LIN {X 0.037,Y -167.701,Z 831.356,A 0.000,B 0.000,C 90.000,E1 244.101} C_DIS
LIN {X 0.050,Y -166.387,Z 831.347,A 0.000,B 0.000,C 90.000,E1 242.359} C_DIS
LIN {X 0.041,Y -163.114,Z 831.327,A 0.000,B 0.000,C 90.000,E1 238.869} C_DIS
LIN {X 0.091,Y -161.064,Z 831.313,A 0.000,B 0.000,C 90.000,E1 236.215} C_DIS
LIN {X -0.021,Y -157.797,Z 831.293,A 0.000,B 0.000,C 90.000,E1 232.718} C_DIS
LIN {X 0.017,Y -155.833,Z 831.278,A 0.000,B 0.000,C 90.000,E1 230.033} C_DIS
LIN {X -0.026,Y -152.084,Z 831.253,A 0.000,B 0.000,C 90.000,E1 225.567} C_DIS
LIN {X -0.007,Y -150.334,Z 831.238,A 0.000,B 0.000,C 90.000,E1 222.852} C_DIS
LIN {X 0.014,Y -147.073,Z 831.213,A 0.000,B 0.000,C 90.000,E1 218.302} C_DIS
LIN {X -0.083,Y -145.648,Z 831.198,A 0.000,B 0.000,C 90.000,E1 215.598} C_DIS
LIN {X -0.078,Y -143.030,Z 831.172,A 0.000,B 0.000,C 90.000,E1 211.003} C_DIS
LIN {X 0.049,Y -141.656,Z 831.152,A 0.000,B 0.000,C 90.000,E1 207.257} C_DIS
LIN {X -0.032,Y -139.446,Z 831.115,A 0.000,B 0.000,C 90.000,E1 200.791} C_DIS
LIN {X 0.021,Y -139.179,Z 831.105,A 0.000,B 0.000,C 90.000,E1 198.906} C_DIS
LIN {X 0.049,Y -138.320,Z 831.053,A 0.000,B 0.000,C 90.000,E1 189.557} C_DIS
LIN {X 0.058,Y -139.466,Z 831.006,A 0.000,B 0.000,C 90.000,E1 181.146} C_DIS
LIN {X 0.000,Y -141.031,Z 830.975,A 0.000,B 0.000,C 90.000,E1 175.584} C_DIS
LIN {X -0.047,Y -142.398,Z 830.960,A 0.000,B 0.000,C 90.000,E1 172.818} C_DIS
LIN {X 0.016,Y -144.630,Z 830.934,A 0.000,B 0.000,C 90.000,E1 168.173} C_DIS
LIN {X 0.076,Y -147.825,Z 830.909,A 0.000,B 0.000,C 90.000,E1 163.559} C_DIS
LIN {X 0.021,Y -150.518,Z 830.889,A 0.000,B 0.000,C 90.000,E1 159.934} C_DIS
LIN {X 0.041,Y -153.979,Z 830.868,A 0.000,B 0.000,C 90.000,E1 156.305} C_DIS
LIN {X -0.038,Y -157.392,Z 830.849,A 0.000,B 0.000,C 90.000,E1 152.743} C_DIS
LIN {X 0.042,Y -161.596,Z 830.829,A 0.000,B 0.000,C 90.000,E1 149.154} C_DIS
LIN {X -0.086,Y -165.793,Z 830.809,A 0.000,B 0.000,C 90.000,E1 145.674} C_DIS
LIN {X 0.034,Y -170.757,Z 830.790,A 0.000,B 0.000,C 90.000,E1 142.145} C_DIS
LIN {X 0.057,Y -175.628,Z 830.771,A 0.000,B 0.000,C 90.000,E1 138.690} C_DIS
LIN {X -0.074,Y -181.244,Z 830.752,A 0.000,B 0.000,C 90.000,E1 135.324} C_DIS
LIN {X 0.057,Y -186.714,Z 830.733,A 0.000,B 0.000,C 90.000,E1 131.919} C_DIS
LIN {X 0.008,Y -191.313,Z 830.719,A 0.000,B 0.000,C 90.000,E1 129.439} C_DIS
LIN {X -0.064,Y -192.836,Z 830.714,A 0.000,B 0.000,C 90.000,E1 128.543} C_DIS
LIN {X -0.132,Y -292.864,Z 830.714,A 0.000,B 0.000,C 90.000,E1 128.543} C_DIS
LIN {X 0.072,Y -295.448,Z 830.714,A 0.000,B 0.000,C 90.000,E1 128.463} C_DIS
LIN {X -0.036,Y -301.314,Z 830.712,A 0.000,B 0.000,C 90.000,E1 128.141} C_DIS
LIN {X -0.096,Y -304.356,Z 830.710,A 0.000,B 0.000,C 90.000,E1 127.810} C_DIS
LIN {X -0.033,Y -306.345,Z 830.708,A 0.000,B 0.000,C 90.000,E1 127.488} C_DIS
LIN {X 0.087,Y -307.898,Z 830.707,A 0.000,B 0.000,C 90.000,E1 127.156} C_DIS
LIN {X -0.132,Y -309.196,Z 830.705,A 0.000,B 0.000,C 90.000,E1 126.870} C_DIS
LIN {X 0.029,Y -321.363,Z 830.683,A 0.000,B 0.000,C 90.000,E1 122.959} C_DIS
LIN {X -0.104,Y -331.880,Z 830.667,A 0.000,B 0.000,C 90.000,E1 120.129} C_DIS
LIN {X 0.017,Y -343.755,Z 830.652,A 0.000,B 0.000,C 90.000,E1 117.308} C_DIS
LIN {X -0.150,Y -357.097,Z 830.636,A 0.000,B 0.000,C 90.000,E1 114.591} C_DIS
LIN {X -0.166,Y -370.281,Z 830.623,A 0.000,B 0.000,C 90.000,E1 112.206} C_DIS
LIN {X 0.217,Y -384.810,Z 830.610,A 0.000,B 0.000,C 90.000,E1 109.812} C_DIS
LIN {X -0.143,Y -400.790,Z 830.598,A 0.000,B 0.000,C 90.000,E1 107.583} C_DIS
LIN {X -0.242,Y -418.334,Z 830.585,A 0.000,B 0.000,C 90.000,E1 105.371} C_DIS
LIN {X -0.002,Y -437.542,Z 830.573,A 0.000,B 0.000,C 90.000,E1 103.175} C_DIS
LIN {X 0.205,Y -457.699,Z 830.562,A 0.000,B 0.000,C 90.000,E1 101.130} C_DIS
LIN {X 0.102,Y -467.922,Z 830.557,A 0.000,B 0.000,C 90.000,E1 100.197} C_DIS
LIN {X 0.100,Y -469.931,Z 830.555,A 0.000,B 0.000,C 90.000,E1 99.962} C_DIS
LIN {X 0.096,Y -471.458,Z 830.554,A 0.000,B 0.000,C 90.000,E1 99.726} C_DIS
LIN {X -0.129,Y -472.703,Z 830.553,A 0.000,B 0.000,C 90.000,E1 99.500} C_DIS
LIN {X 0.193,Y -473.614,Z 830.551,A 0.000,B 0.000,C 90.000,E1 99.208} C_DIS
LIN {X -0.161,Y -474.606,Z 830.548,A 0.000,B 0.000,C 90.000,E1 98.746} C_DIS
LIN {X 0.031,Y -474.616,Z 830.546,A 0.000,B 0.000,C 90.000,E1 98.219} C_DIS
LIN {X 0.158,Y -473.647,Z 830.543,A 0.000,B 0.000,C 90.000,E1 97.701} C_DIS
LIN {X -0.182,Y -471.537,Z 830.540,A 0.000,B 0.000,C 90.000,E1 97.239} C_DIS
LIN {X -0.007,Y -453.828,Z 830.525,A 0.000,B 0.000,C 90.000,E1 94.416} C_DIS
LIN {X 0.139,Y -443.235,Z 830.514,A 0.000,B 0.000,C 90.000,E1 92.579} C_DIS
LIN {X -0.113,Y -433.972,Z 830.506,A 0.000,B 0.000,C 90.000,E1 91.031} C_DIS
LIN {X 0.194,Y -425.976,Z 830.498,A 0.000,B 0.000,C 90.000,E1 89.656} C_DIS
LIN {X 0.177,Y -414.567,Z 830.488,A 0.000,B 0.000,C 90.000,E1 87.764} C_DIS
LIN {X -0.138,Y -404.693,Z 830.479,A 0.000,B 0.000,C 90.000,E1 86.159} C_DIS
LIN {X -0.074,Y -391.516,Z 830.466,A 0.000,B 0.000,C 90.000,E1 83.913} C_DIS
LIN {X 0.083,Y -380.237,Z 830.455,A 0.000,B 0.000,C 90.000,E1 81.894} C_DIS
LIN {X 0.026,Y -366.068,Z 830.440,A 0.000,B 0.000,C 90.000,E1 79.285} C_DIS
LIN {X -0.146,Y -354.091,Z 830.427,A 0.000,B 0.000,C 90.000,E1 76.937} C_DIS
LIN {X -0.092,Y -343.657,Z 830.416,A 0.000,B 0.000,C 90.000,E1 74.810} C_DIS
LIN {X 0.123,Y -331.831,Z 830.402,A 0.000,B 0.000,C 90.000,E1 72.308} C_DIS
LIN {X 0.090,Y -321.680,Z 830.390,A 0.000,B 0.000,C 90.000,E1 70.115} C_DIS
LIN {X 0.006,Y -307.585,Z 830.372,A 0.000,B 0.000,C 90.000,E1 66.922} C_DIS
LIN {X -0.030,Y -295.560,Z 830.355,A 0.000,B 0.000,C 90.000,E1 63.973} C_DIS
LIN {X -0.105,Y -285.303,Z 830.340,A 0.000,B 0.000,C 90.000,E1 61.307} C_DIS
LIN {X -0.018,Y -272.949,Z 830.321,A 0.000,B 0.000,C 90.000,E1 57.867} C_DIS
LIN {X 0.025,Y -261.379,Z 830.302,A 0.000,B 0.000,C 90.000,E1 54.356} C_DIS
LIN {X -0.119,Y -251.415,Z 830.284,A 0.000,B 0.000,C 90.000,E1 51.170} C_DIS
LIN {X 0.123,Y -240.989,Z 830.264,A 0.000,B 0.000,C 90.000,E1 47.472} C_DIS
LIN {X -0.005,Y -231.404,Z 830.243,A 0.000,B 0.000,C 90.000,E1 43.785} C_DIS
LIN {X -0.098,Y -224.188,Z 830.226,A 0.000,B 0.000,C 90.000,E1 40.782} C_DIS
LIN {X 0.001,Y -217.178,Z 830.209,A 0.000,B 0.000,C 90.000,E1 37.684} C_DIS
LIN {X 0.007,Y -210.622,Z 830.192,A 0.000,B 0.000,C 90.000,E1 34.565} C_DIS
LIN {X 0.062,Y -203.042,Z 830.170,A 0.000,B 0.000,C 90.000,E1 30.590} C_DIS
LIN {X 0.034,Y -197.729,Z 830.152,A 0.000,B 0.000,C 90.000,E1 27.385} C_DIS
LIN {X 0.044,Y -193.102,Z 830.134,A 0.000,B 0.000,C 90.000,E1 24.131} C_DIS
LIN {X -0.012,Y -189.298,Z 830.116,A 0.000,B 0.000,C 90.000,E1 20.865} C_DIS
LIN {X -0.044,Y -185.602,Z 830.093,A 0.000,B 0.000,C 90.000,E1 16.732} C_DIS
LIN {X -0.030,Y -182.647,Z 830.065,A 0.000,B 0.000,C 90.000,E1 11.715} C_DIS
LIN {X -0.009,Y -183.562,Z 829.969,A 0.000,B 0.000,C 90.000,E1 354.489} C_DIS
LIN {X 0.045,Y -186.904,Z 829.941,A 0.000,B 0.000,C 90.000,E1 349.454} C_DIS
LIN {X -0.069,Y -190.678,Z 829.918,A 0.000,B 0.000,C 90.000,E1 345.338} C_DIS
LIN {X -0.059,Y -195.359,Z 829.896,A 0.000,B 0.000,C 90.000,E1 341.221} C_DIS
LIN {X 0.111,Y -200.918,Z 829.873,A 0.000,B 0.000,C 90.000,E1 337.102} C_DIS
LIN {X -0.043,Y -207.259,Z 829.851,A 0.000,B 0.000,C 90.000,E1 333.127} C_DIS
LIN {X -0.001,Y -214.528,Z 829.829,A 0.000,B 0.000,C 90.000,E1 329.154} C_DIS
LIN {X -0.026,Y -222.613,Z 829.807,A 0.000,B 0.000,C 90.000,E1 325.261} C_DIS
LIN {X 0.045,Y -231.613,Z 829.786,A 0.000,B 0.000,C 90.000,E1 321.412} C_DIS
LIN {X -0.033,Y -241.736,Z 829.765,A 0.000,B 0.000,C 90.000,E1 317.676} C_DIS
LIN {X 0.031,Y -251.698,Z 829.746,A 0.000,B 0.000,C 90.000,E1 314.352} C_DIS
LIN {X -0.151,Y -262.548,Z 829.728,A 0.000,B 0.000,C 90.000,E1 311.148} C_DIS
LIN {X 0.030,Y -274.288,Z 829.711,A 0.000,B 0.000,C 90.000,E1 307.935} C_DIS
LIN {X 0.100,Y -286.955,Z 829.694,A 0.000,B 0.000,C 90.000,E1 304.818} C_DIS
LIN {X 0.070,Y -302.514,Z 829.675,A 0.000,B 0.000,C 90.000,E1 301.465} C_DIS
LIN {X -0.067,Y -316.280,Z 829.660,A 0.000,B 0.000,C 90.000,E1 298.871} C_DIS
LIN {X 0.074,Y -327.632,Z 829.650,A 0.000,B 0.000,C 90.000,E1 296.924} C_DIS
LIN {X -0.035,Y -347.921,Z 829.632,A 0.000,B 0.000,C 90.000,E1 293.823} C_DIS
LIN {X 0.017,Y -368.274,Z 829.617,A 0.000,B 0.000,C 90.000,E1 291.099} C_DIS
LIN {X 0.106,Y -393.423,Z 829.601,A 0.000,B 0.000,C 90.000,E1 288.181} C_DIS
LIN {X 0.047,Y -406.328,Z 829.593,A 0.000,B 0.000,C 90.000,E1 286.804} C_DIS
LIN {X -0.149,Y -418.954,Z 829.586,A 0.000,B 0.000,C 90.000,E1 285.481} C_DIS
LIN {X -0.148,Y -428.903,Z 829.580,A 0.000,B 0.000,C 90.000,E1 284.411} C_DIS
LIN {X -0.027,Y -441.051,Z 829.573,A 0.000,B 0.000,C 90.000,E1 283.063} C_DIS
LIN {X -0.013,Y -450.318,Z 829.567,A 0.000,B 0.000,C 90.000,E1 282.007} C_DIS
LIN {X 0.108,Y -459.010,Z 829.561,A 0.000,B 0.000,C 90.000,E1 280.950} C_DIS
LIN {X -0.211,Y -467.084,Z 829.555,A 0.000,B 0.000,C 90.000,E1 279.962} C_DIS
LIN {X 0.173,Y -472.643,Z 829.551,A 0.000,B 0.000,C 90.000,E1 279.151} C_DIS
LIN {X 0.140,Y -477.681,Z 829.547,A 0.000,B 0.000,C 90.000,E1 278.398} C_DIS
LIN {X 0.155,Y -481.989,Z 829.543,A 0.000,B 0.000,C 90.000,E1 277.644} C_DIS
LIN {X 0.200,Y -485.646,Z 829.538,A 0.000,B 0.000,C 90.000,E1 276.891} C_DIS
LIN {X -0.093,Y -487.710,Z 829.536,A 0.000,B 0.000,C 90.000,E1 276.429} C_DIS
LIN {X 0.109,Y -489.419,Z 829.533,A 0.000,B 0.000,C 90.000,E1 275.910} C_DIS
LIN {X -0.171,Y -490.752,Z 829.530,A 0.000,B 0.000,C 90.000,E1 275.448} C_DIS
LIN {X 0.004,Y -491.765,Z 829.527,A 0.000,B 0.000,C 90.000,E1 274.935} C_DIS
LIN {X 0.232,Y -492.413,Z 829.525,A 0.000,B 0.000,C 90.000,E1 274.416} C_DIS
LIN {X -0.029,Y -492.738,Z 829.522,A 0.000,B 0.000,C 90.000,E1 273.955} C_DIS
LIN {X 0.172,Y -492.604,Z 829.519,A 0.000,B 0.000,C 90.000,E1 273.440} C_DIS
LIN {X -0.087,Y -492.130,Z 829.516,A 0.000,B 0.000,C 90.000,E1 272.980} C_DIS
LIN {X 0.119,Y -491.281,Z 829.514,A 0.000,B 0.000,C 90.000,E1 272.465} C_DIS
LIN {X -0.165,Y -489.925,Z 829.511,A 0.000,B 0.000,C 90.000,E1 272.007} C_DIS
LIN {X 0.051,Y -488.177,Z 829.508,A 0.000,B 0.000,C 90.000,E1 271.489} C_DIS
LIN {X 0.242,Y -485.870,Z 829.506,A 0.000,B 0.000,C 90.000,E1 270.974} C_DIS
LIN {X -0.066,Y -482.988,Z 829.503,A 0.000,B 0.000,C 90.000,E1 270.516} C_DIS
LIN {X 0.096,Y -479.459,Z 829.500,A 0.000,B 0.000,C 90.000,E1 270.000} C_DIS
LIN {X 0.237,Y -475.133,Z 829.497,A 0.000,B 0.000,C 90.000,E1 269.484} C_DIS
LIN {X -0.118,Y -469.908,Z 829.495,A 0.000,B 0.000,C 90.000,E1 269.026} C_DIS
LIN {X -0.174,Y -463.953,Z 829.492,A 0.000,B 0.000,C 90.000,E1 268.568} C_DIS
LIN {X 0.033,Y -460.941,Z 829.491,A 0.000,B 0.000,C 90.000,E1 268.339} C_DIS
LIN {X -0.206,Y -457.485,Z 829.490,A 0.000,B 0.000,C 90.000,E1 268.165} C_DIS
LIN {X -0.179,Y -450.261,Z 829.488,A 0.000,B 0.000,C 90.000,E1 267.822} C_DIS
LIN {X -0.036,Y -442.707,Z 829.486,A 0.000,B 0.000,C 90.000,E1 267.535} C_DIS
LIN {X 0.129,Y -434.241,Z 829.485,A 0.000,B 0.000,C 90.000,E1 267.306} C_DIS
LIN {X -0.058,Y -424.909,Z 829.484,A 0.000,B 0.000,C 90.000,E1 267.192} C_DIS
LIN {X 0.113,Y -420.260,Z 829.484,A 0.000,B 0.000,C 90.000,E1 267.135} C_DIS
LIN {X 0.029,Y -414.526,Z 829.484,A 0.000,B 0.000,C 90.000,E1 267.135} C_DIS
LIN {X -0.023,Y -181.005,Z 829.484,A 0.000,B 0.000,C 90.000,E1 267.135} C_DIS
LIN {X -0.014,Y -180.907,Z 829.474,A 0.000,B 0.000,C 90.000,E1 265.412} C_DIS
LIN {X 0.042,Y -180.707,Z 829.470,A 0.000,B 0.000,C 90.000,E1 264.552} C_DIS
LIN {X -0.040,Y -178.794,Z 829.442,A 0.000,B 0.000,C 90.000,E1 259.511} C_DIS
LIN {X 0.038,Y -175.840,Z 829.413,A 0.000,B 0.000,C 90.000,E1 254.393} C_DIS
LIN {X 0.038,Y -172.030,Z 829.385,A 0.000,B 0.000,C 90.000,E1 249.263} C_DIS
LIN {X 0.014,Y -171.458,Z 829.380,A 0.000,B 0.000,C 90.000,E1 248.411} C_DIS
LIN {X -0.006,Y -167.691,Z 829.356,A 0.000,B 0.000,C 90.000,E1 244.101} C_DIS
LIN {X 0.007,Y -166.373,Z 829.346,A 0.000,B 0.000,C 90.000,E1 242.359} C_DIS
LIN {X 0.000,Y -163.103,Z 829.327,A 0.000,B 0.000,C 90.000,E1 238.869} C_DIS
LIN {X 0.050,Y -161.049,Z 829.312,A 0.000,B 0.000,C 90.000,E1 236.215} C_DIS
LIN {X 0.033,Y -157.786,Z 829.293,A 0.000,B 0.000,C 90.000,E1 232.683} C_DIS
LIN {X -0.024,Y -155.822,Z 829.278,A 0.000,B 0.000,C 90.000,E1 230.033} C_DIS
LIN {X -0.066,Y -152.073,Z 829.253,A 0.000,B 0.000,C 90.000,E1 225.567} C_DIS
LIN {X -0.047,Y -150.323,Z 829.238,A 0.000,B 0.000,C 90.000,E1 222.852} C_DIS
LIN {X -0.025,Y -147.065,Z 829.213,A 0.000,B 0.000,C 90.000,E1 218.302} C_DIS
LIN {X 0.083,Y -145.641,Z 829.198,A 0.000,B 0.000,C 90.000,E1 215.518} C_DIS
LIN {X 0.080,Y -143.023,Z 829.172,A 0.000,B 0.000,C 90.000,E1 210.924} C_DIS
LIN {X 0.011,Y -141.649,Z 829.151,A 0.000,B 0.000,C 90.000,E1 207.257} C_DIS
LIN {X 0.061,Y -139.442,Z 829.115,A 0.000,B 0.000,C 90.000,E1 200.737} C_DIS
LIN {X -0.017,Y -139.176,Z 829.105,A 0.000,B 0.000,C 90.000,E1 198.906} C_DIS
LIN {X 0.011,Y -138.318,Z 829.053,A 0.000,B 0.000,C 90.000,E1 189.557} C_DIS
LIN {X 0.021,Y -139.469,Z 829.006,A 0.000,B 0.000,C 90.000,E1 181.146} C_DIS
LIN {X -0.039,Y -141.038,Z 828.975,A 0.000,B 0.000,C 90.000,E1 175.584} C_DIS
LIN {X 0.056,Y -142.406,Z 828.960,A 0.000,B 0.000,C 90.000,E1 172.761} C_DIS
LIN {X -0.023,Y -144.639,Z 828.934,A 0.000,B 0.000,C 90.000,E1 168.173} C_DIS
LIN {X 0.036,Y -147.835,Z 828.909,A 0.000,B 0.000,C 90.000,E1 163.559} C_DIS
LIN {X -0.019,Y -150.530,Z 828.888,A 0.000,B 0.000,C 90.000,E1 159.934} C_DIS
LIN {X 0.000,Y -153.994,Z 828.868,A 0.000,B 0.000,C 90.000,E1 156.305} C_DIS
LIN {X -0.079,Y -157.407,Z 828.848,A 0.000,B 0.000,C 90.000,E1 152.743} C_DIS
LIN {X 0.000,Y -161.615,Z 828.829,A 0.000,B 0.000,C 90.000,E1 149.154} C_DIS
LIN {X 0.102,Y -165.812,Z 828.809,A 0.000,B 0.000,C 90.000,E1 145.595} C_DIS
LIN {X -0.009,Y -170.779,Z 828.790,A 0.000,B 0.000,C 90.000,E1 142.145} C_DIS
LIN {X 0.012,Y -175.650,Z 828.771,A 0.000,B 0.000,C 90.000,E1 138.690} C_DIS
LIN {X 0.011,Y -181.264,Z 828.752,A 0.000,B 0.000,C 90.000,E1 135.283} C_DIS
LIN {X 0.011,Y -186.739,Z 828.733,A 0.000,B 0.000,C 90.000,E1 131.919} C_DIS
LIN {X -0.038,Y -191.336,Z 828.719,A 0.000,B 0.000,C 90.000,E1 129.439} C_DIS
LIN {X -0.040,Y -192.824,Z 828.714,A 0.000,B 0.000,C 90.000,E1 128.543} C_DIS
LIN {X -0.096,Y -293.128,Z 828.714,A 0.000,B 0.000,C 90.000,E1 128.543} C_DIS
LIN {X 0.002,Y -296.105,Z 828.714,A 0.000,B 0.000,C 90.000,E1 128.463} C_DIS
LIN {X 0.129,Y -301.507,Z 828.712,A 0.000,B 0.000,C 90.000,E1 128.096} C_DIS
LIN {X -0.168,Y -304.472,Z 828.710,A 0.000,B 0.000,C 90.000,E1 127.810} C_DIS
LIN {X 0.106,Y -306.456,Z 828.708,A 0.000,B 0.000,C 90.000,E1 127.443} C_DIS
LIN {X -0.049,Y -308.003,Z 828.706,A 0.000,B 0.000,C 90.000,E1 127.156} C_DIS
LIN {X 0.164,Y -309.268,Z 828.705,A 0.000,B 0.000,C 90.000,E1 126.790} C_DIS
LIN {X -0.111,Y -321.427,Z 828.683,A 0.000,B 0.000,C 90.000,E1 122.959} C_DIS
LIN {X 0.041,Y -331.956,Z 828.667,A 0.000,B 0.000,C 90.000,E1 120.079} C_DIS
LIN {X 0.178,Y -343.842,Z 828.652,A 0.000,B 0.000,C 90.000,E1 117.257} C_DIS
LIN {X 0.175,Y -357.197,Z 828.636,A 0.000,B 0.000,C 90.000,E1 114.515} C_DIS
LIN {X 0.026,Y -370.394,Z 828.623,A 0.000,B 0.000,C 90.000,E1 112.153} C_DIS
LIN {X 0.063,Y -384.938,Z 828.610,A 0.000,B 0.000,C 90.000,E1 109.812} C_DIS
LIN {X 0.202,Y -400.932,Z 828.597,A 0.000,B 0.000,C 90.000,E1 107.511} C_DIS
LIN {X 0.002,Y -418.492,Z 828.585,A 0.000,B 0.000,C 90.000,E1 105.315} C_DIS
LIN {X -0.163,Y -437.714,Z 828.573,A 0.000,B 0.000,C 90.000,E1 103.175} C_DIS
LIN {X 0.048,Y -457.877,Z 828.562,A 0.000,B 0.000,C 90.000,E1 101.130} C_DIS
LIN {X -0.052,Y -468.080,Z 828.557,A 0.000,B 0.000,C 90.000,E1 100.197} C_DIS
LIN {X -0.064,Y -470.061,Z 828.555,A 0.000,B 0.000,C 90.000,E1 99.962} C_DIS
LIN {X -0.077,Y -471.568,Z 828.554,A 0.000,B 0.000,C 90.000,E1 99.726} C_DIS
LIN {X 0.165,Y -472.786,Z 828.553,A 0.000,B 0.000,C 90.000,E1 99.443} C_DIS
LIN {X 0.019,Y -473.678,Z 828.551,A 0.000,B 0.000,C 90.000,E1 99.208} C_DIS
LIN {X 0.136,Y -474.635,Z 828.548,A 0.000,B 0.000,C 90.000,E1 98.690} C_DIS
LIN {X -0.142,Y -474.611,Z 828.546,A 0.000,B 0.000,C 90.000,E1 98.219} C_DIS
LIN {X -0.014,Y -473.607,Z 828.543,A 0.000,B 0.000,C 90.000,E1 97.701} C_DIS
LIN {X 0.115,Y -471.453,Z 828.540,A 0.000,B 0.000,C 90.000,E1 97.182} C_DIS
LIN {X -0.174,Y -453.736,Z 828.524,A 0.000,B 0.000,C 90.000,E1 94.416} C_DIS
LIN {X 0.158,Y -441.632,Z 828.513,A 0.000,B 0.000,C 90.000,E1 92.293} C_DIS
LIN {X -0.121,Y -432.309,Z 828.504,A 0.000,B 0.000,C 90.000,E1 90.745} C_DIS
LIN {X -0.133,Y -422.637,Z 828.495,A 0.000,B 0.000,C 90.000,E1 89.141} C_DIS
LIN {X 0.199,Y -411.221,Z 828.485,A 0.000,B 0.000,C 90.000,E1 87.192} C_DIS
LIN {X -0.104,Y -399.640,Z 828.474,A 0.000,B 0.000,C 90.000,E1 85.298} C_DIS
LIN {X -0.117,Y -384.964,Z 828.460,A 0.000,B 0.000,C 90.000,E1 82.761} C_DIS
LIN {X -0.039,Y -369.097,Z 828.444,A 0.000,B 0.000,C 90.000,E1 79.859} C_DIS
LIN {X 0.099,Y -355.518,Z 828.429,A 0.000,B 0.000,C 90.000,E1 77.173} C_DIS
LIN {X 0.181,Y -345.086,Z 828.417,A 0.000,B 0.000,C 90.000,E1 75.046} C_DIS
LIN {X 0.121,Y -334.736,Z 828.405,A 0.000,B 0.000,C 90.000,E1 72.906} C_DIS
LIN {X -0.002,Y -323.108,Z 828.391,A 0.000,B 0.000,C 90.000,E1 70.423} C_DIS
LIN {X -0.040,Y -308.981,Z 828.373,A 0.000,B 0.000,C 90.000,E1 67.230} C_DIS
LIN {X -0.027,Y -296.924,Z 828.357,A 0.000,B 0.000,C 90.000,E1 64.280} C_DIS
LIN {X -0.050,Y -287.940,Z 828.344,A 0.000,B 0.000,C 90.000,E1 61.948} C_DIS
LIN {X 0.078,Y -277.942,Z 828.329,A 0.000,B 0.000,C 90.000,E1 59.203} C_DIS
LIN {X -0.019,Y -266.142,Z 828.310,A 0.000,B 0.000,C 90.000,E1 55.754} C_DIS
LIN {X -0.025,Y -257.170,Z 828.294,A 0.000,B 0.000,C 90.000,E1 52.924} C_DIS
LIN {X 0.048,Y -247.442,Z 828.276,A 0.000,B 0.000,C 90.000,E1 49.666} C_DIS
LIN {X 0.141,Y -237.335,Z 828.256,A 0.000,B 0.000,C 90.000,E1 45.972} C_DIS
LIN {X -0.095,Y -228.056,Z 828.235,A 0.000,B 0.000,C 90.000,E1 42.285} C_DIS
LIN {X 0.066,Y -220.977,Z 828.218,A 0.000,B 0.000,C 90.000,E1 39.197} C_DIS
LIN {X 0.112,Y -214.125,Z 828.201,A 0.000,B 0.000,C 90.000,E1 36.091} C_DIS
LIN {X -0.073,Y -206.282,Z 828.179,A 0.000,B 0.000,C 90.000,E1 32.212} C_DIS
LIN {X 0.006,Y -200.574,Z 828.161,A 0.000,B 0.000,C 90.000,E1 28.999} C_DIS
LIN {X 0.020,Y -194.496,Z 828.139,A 0.000,B 0.000,C 90.000,E1 24.951} C_DIS
LIN {X 0.069,Y -190.478,Z 828.120,A 0.000,B 0.000,C 90.000,E1 21.663} C_DIS
LIN {X -0.102,Y -186.534,Z 828.098,A 0.000,B 0.000,C 90.000,E1 17.583} C_DIS
LIN {X 0.044,Y -183.328,Z 828.070,A 0.000,B 0.000,C 90.000,E1 12.535} C_DIS
LIN {X 0.051,Y -181.292,Z 828.023,A 0.000,B 0.000,C 90.000,E1 4.131} C_DIS
LIN {X 0.028,Y -183.049,Z 827.979,A 0.000,B 0.000,C 90.000,E1 356.159} C_DIS
LIN {X 0.007,Y -185.940,Z 827.951,A 0.000,B 0.000,C 90.000,E1 351.141} C_DIS
LIN {X -0.061,Y -190.112,Z 827.923,A 0.000,B 0.000,C 90.000,E1 346.172} C_DIS
LIN {X -0.068,Y -194.590,Z 827.900,A 0.000,B 0.000,C 90.000,E1 342.054} C_DIS
LIN {X -0.061,Y -199.950,Z 827.878,A 0.000,B 0.000,C 90.000,E1 337.975} C_DIS
LIN {X -0.062,Y -206.117,Z 827.855,A 0.000,B 0.000,C 90.000,E1 333.948} C_DIS
LIN {X 0.033,Y -213.211,Z 827.833,A 0.000,B 0.000,C 90.000,E1 329.950} C_DIS
LIN {X -0.152,Y -221.116,Z 827.811,A 0.000,B 0.000,C 90.000,E1 326.087} C_DIS
LIN {X 0.055,Y -229.927,Z 827.790,A 0.000,B 0.000,C 90.000,E1 322.190} C_DIS
LIN {X 0.151,Y -238.804,Z 827.771,A 0.000,B 0.000,C 90.000,E1 318.771} C_DIS
LIN {X -0.045,Y -248.401,Z 827.753,A 0.000,B 0.000,C 90.000,E1 315.486} C_DIS
LIN {X 0.033,Y -259.000,Z 827.734,A 0.000,B 0.000,C 90.000,E1 312.204} C_DIS
LIN {X -0.099,Y -270.344,Z 827.717,A 0.000,B 0.000,C 90.000,E1 309.036} C_DIS
LIN {X 0.022,Y -282.614,Z 827.699,A 0.000,B 0.000,C 90.000,E1 305.884} C_DIS
LIN {X 0.015,Y -297.636,Z 827.681,A 0.000,B 0.000,C 90.000,E1 302.498} C_DIS
LIN {X -0.041,Y -312.648,Z 827.664,A 0.000,B 0.000,C 90.000,E1 299.539} C_DIS
LIN {X 0.034,Y -323.611,Z 827.653,A 0.000,B 0.000,C 90.000,E1 297.590} C_DIS
LIN {X -0.145,Y -337.381,Z 827.641,A 0.000,B 0.000,C 90.000,E1 295.412} C_DIS
LIN {X 0.134,Y -352.063,Z 827.629,A 0.000,B 0.000,C 90.000,E1 293.206} C_DIS
LIN {X -0.118,Y -370.414,Z 827.616,A 0.000,B 0.000,C 90.000,E1 290.844} C_DIS
LIN {X -0.094,Y -395.688,Z 827.600,A 0.000,B 0.000,C 90.000,E1 287.946} C_DIS
LIN {X -0.005,Y -408.557,Z 827.592,A 0.000,B 0.000,C 90.000,E1 286.551} C_DIS
LIN {X 0.074,Y -421.192,Z 827.584,A 0.000,B 0.000,C 90.000,E1 285.190} C_DIS
LIN {X 0.075,Y -433.245,Z 827.577,A 0.000,B 0.000,C 90.000,E1 283.883} C_DIS
LIN {X -0.005,Y -442.952,Z 827.571,A 0.000,B 0.000,C 90.000,E1 282.827} C_DIS
LIN {X 0.030,Y -452.071,Z 827.565,A 0.000,B 0.000,C 90.000,E1 281.771} C_DIS
LIN {X 0.085,Y -460.685,Z 827.560,A 0.000,B 0.000,C 90.000,E1 280.725} C_DIS
LIN {X -0.131,Y -468.609,Z 827.554,A 0.000,B 0.000,C 90.000,E1 279.726} C_DIS
LIN {X -0.207,Y -474.003,Z 827.550,A 0.000,B 0.000,C 90.000,E1 278.973} C_DIS
LIN {X 0.243,Y -478.848,Z 827.546,A 0.000,B 0.000,C 90.000,E1 278.163} C_DIS
LIN {X 0.261,Y -483.011,Z 827.541,A 0.000,B 0.000,C 90.000,E1 277.409} C_DIS
LIN {X -0.223,Y -486.508,Z 827.537,A 0.000,B 0.000,C 90.000,E1 276.720} C_DIS
LIN {X 0.141,Y -487.533,Z 827.536,A 0.000,B 0.000,C 90.000,E1 276.429} C_DIS
LIN {X -0.143,Y -489.264,Z 827.533,A 0.000,B 0.000,C 90.000,E1 275.967} C_DIS
LIN {X 0.017,Y -490.629,Z 827.530,A 0.000,B 0.000,C 90.000,E1 275.454} C_DIS
LIN {X -0.252,Y -491.683,Z 827.528,A 0.000,B 0.000,C 90.000,E1 274.992} C_DIS
LIN {X -0.026,Y -492.373,Z 827.525,A 0.000,B 0.000,C 90.000,E1 274.473} C_DIS
LIN {X 0.204,Y -492.716,Z 827.522,A 0.000,B 0.000,C 90.000,E1 273.955} C_DIS
LIN {X -0.087,Y -492.648,Z 827.519,A 0.000,B 0.000,C 90.000,E1 273.498} C_DIS
LIN {X 0.145,Y -492.193,Z 827.517,A 0.000,B 0.000,C 90.000,E1 272.980} C_DIS
LIN {X -0.140,Y -491.339,Z 827.514,A 0.000,B 0.000,C 90.000,E1 272.522} C_DIS
LIN {X 0.067,Y -490.065,Z 827.511,A 0.000,B 0.000,C 90.000,E1 272.007} C_DIS
LIN {X -0.205,Y -488.373,Z 827.508,A 0.000,B 0.000,C 90.000,E1 271.547} C_DIS
LIN {X -0.012,Y -486.127,Z 827.506,A 0.000,B 0.000,C 90.000,E1 271.031} C_DIS
LIN {X 0.165,Y -483.328,Z 827.503,A 0.000,B 0.000,C 90.000,E1 270.516} C_DIS
LIN {X -0.153,Y -479.875,Z 827.500,A 0.000,B 0.000,C 90.000,E1 270.057} C_DIS
LIN {X -0.007,Y -475.644,Z 827.497,A 0.000,B 0.000,C 90.000,E1 269.542} C_DIS
LIN {X 0.113,Y -470.545,Z 827.495,A 0.000,B 0.000,C 90.000,E1 269.026} C_DIS
LIN {X -0.019,Y -464.626,Z 827.492,A 0.000,B 0.000,C 90.000,E1 268.568} C_DIS
LIN {X 0.142,Y -461.589,Z 827.491,A 0.000,B 0.000,C 90.000,E1 268.339} C_DIS
LIN {X -0.137,Y -454.775,Z 827.489,A 0.000,B 0.000,C 90.000,E1 267.993} C_DIS
LIN {X 0.154,Y -447.481,Z 827.487,A 0.000,B 0.000,C 90.000,E1 267.650} C_DIS
LIN {X 0.049,Y -439.815,Z 827.486,A 0.000,B 0.000,C 90.000,E1 267.421} C_DIS
LIN {X -0.017,Y -431.207,Z 827.485,A 0.000,B 0.000,C 90.000,E1 267.249} C_DIS
LIN {X -0.141,Y -425.903,Z 827.484,A 0.000,B 0.000,C 90.000,E1 267.192} C_DIS
LIN {X -0.096,Y -417.064,Z 827.484,A 0.000,B 0.000,C 90.000,E1 267.135} C_DIS
LIN {X -0.061,Y -181.004,Z 827.484,A 0.000,B 0.000,C 90.000,E1 267.135} C_DIS
LIN {X -0.064,Y -180.907,Z 827.474,A 0.000,B 0.000,C 90.000,E1 265.412} C_DIS
LIN {X 0.011,Y -180.700,Z 827.470,A 0.000,B 0.000,C 90.000,E1 264.546} C_DIS
LIN {X 0.088,Y -178.786,Z 827.442,A 0.000,B 0.000,C 90.000,E1 259.454} C_DIS
LIN {X -0.010,Y -175.832,Z 827.413,A 0.000,B 0.000,C 90.000,E1 254.393} C_DIS
LIN {X -0.009,Y -172.021,Z 827.385,A 0.000,B 0.000,C 90.000,E1 249.263} C_DIS
LIN {X -0.033,Y -171.444,Z 827.380,A 0.000,B 0.000,C 90.000,E1 248.411} C_DIS
LIN {X 0.021,Y -167.679,Z 827.356,A 0.000,B 0.000,C 90.000,E1 244.076} C_DIS
LIN {X -0.038,Y -166.356,Z 827.346,A 0.000,B 0.000,C 90.000,E1 242.359} C_DIS
LIN {X -0.046,Y -163.089,Z 827.327,A 0.000,B 0.000,C 90.000,E1 238.869} C_DIS
LIN {X 0.005,Y -161.033,Z 827.312,A 0.000,B 0.000,C 90.000,E1 236.215} C_DIS
LIN {X -0.011,Y -157.772,Z 827.293,A 0.000,B 0.000,C 90.000,E1 232.683} C_DIS
LIN {X 0.051,Y -155.810,Z 827.278,A 0.000,B 0.000,C 90.000,E1 229.989} C_DIS
LIN {X -0.001,Y -152.061,Z 827.253,A 0.000,B 0.000,C 90.000,E1 225.526} C_DIS
LIN {X 0.012,Y -150.311,Z 827.238,A 0.000,B 0.000,C 90.000,E1 222.813} C_DIS
LIN {X 0.047,Y -147.055,Z 827.213,A 0.000,B 0.000,C 90.000,E1 218.257} C_DIS
LIN {X 0.039,Y -145.633,Z 827.197,A 0.000,B 0.000,C 90.000,E1 215.518} C_DIS
LIN {X 0.038,Y -143.016,Z 827.172,A 0.000,B 0.000,C 90.000,E1 210.924} C_DIS
LIN {X -0.031,Y -141.642,Z 827.151,A 0.000,B 0.000,C 90.000,E1 207.257} C_DIS
LIN {X 0.019,Y -139.439,Z 827.115,A 0.000,B 0.000,C 90.000,E1 200.737} C_DIS
LIN {X -0.058,Y -139.172,Z 827.105,A 0.000,B 0.000,C 90.000,E1 198.906} C_DIS
LIN {X -0.030,Y -138.318,Z 827.053,A 0.000,B 0.000,C 90.000,E1 189.557} C_DIS
LIN {X -0.021,Y -139.471,Z 827.006,A 0.000,B 0.000,C 90.000,E1 181.146} C_DIS
LIN {X 0.060,Y -141.045,Z 826.975,A 0.000,B 0.000,C 90.000,E1 175.527} C_DIS
LIN {X 0.014,Y -142.414,Z 826.960,A 0.000,B 0.000,C 90.000,E1 172.761} C_DIS
LIN {X -0.066,Y -144.649,Z 826.934,A 0.000,B 0.000,C 90.000,E1 168.173} C_DIS
LIN {X -0.006,Y -147.845,Z 826.909,A 0.000,B 0.000,C 90.000,E1 163.559} C_DIS
LIN {X -0.063,Y -150.544,Z 826.888,A 0.000,B 0.000,C 90.000,E1 159.934} C_DIS
LIN {X -0.044,Y -154.011,Z 826.868,A 0.000,B 0.000,C 90.000,E1 156.305} C_DIS
LIN {X 0.016,Y -157.425,Z 826.848,A 0.000,B 0.000,C 90.000,E1 152.692} C_DIS
LIN {X 0.038,Y -161.637,Z 826.829,A 0.000,B 0.000,C 90.000,E1 149.125} C_DIS
LIN {X 0.055,Y -165.833,Z 826.809,A 0.000,B 0.000,C 90.000,E1 145.595} C_DIS
LIN {X 0.048,Y -170.804,Z 826.790,A 0.000,B 0.000,C 90.000,E1 142.110} C_DIS
LIN {X -0.036,Y -175.674,Z 826.770,A 0.000,B 0.000,C 90.000,E1 138.690} C_DIS
LIN {X 0.088,Y -181.288,Z 826.752,A 0.000,B 0.000,C 90.000,E1 135.243} C_DIS
LIN {X -0.039,Y -186.767,Z 826.733,A 0.000,B 0.000,C 90.000,E1 131.919} C_DIS
LIN {X 0.033,Y -191.360,Z 826.719,A 0.000,B 0.000,C 90.000,E1 129.402} C_DIS
LIN {X -0.021,Y -192.814,Z 826.714,A 0.000,B 0.000,C 90.000,E1 128.543} C_DIS
LIN {X -0.084,Y -293.726,Z 826.714,A 0.000,B 0.000,C 90.000,E1 128.543} C_DIS
LIN {X -0.049,Y -298.950,Z 826.713,A 0.000,B 0.000,C 90.000,E1 128.338} C_DIS
LIN {X -0.008,Y -301.349,Z 826.712,A 0.000,B 0.000,C 90.000,E1 128.141} C_DIS
LIN {X 0.178,Y -304.595,Z 826.710,A 0.000,B 0.000,C 90.000,E1 127.729} C_DIS
LIN {X 0.020,Y -306.546,Z 826.708,A 0.000,B 0.000,C 90.000,E1 127.443} C_DIS
LIN {X -0.142,Y -308.068,Z 826.706,A 0.000,B 0.000,C 90.000,E1 127.156} C_DIS
LIN {X 0.072,Y -309.310,Z 826.704,A 0.000,B 0.000,C 90.000,E1 126.790} C_DIS
LIN {X -0.015,Y -320.375,Z 826.685,A 0.000,B 0.000,C 90.000,E1 123.245} C_DIS
LIN {X 0.000,Y -330.763,Z 826.669,A 0.000,B 0.000,C 90.000,E1 120.384} C_DIS
LIN {X -0.074,Y -342.504,Z 826.653,A 0.000,B 0.000,C 90.000,E1 117.590} C_DIS
LIN {X 0.038,Y -355.696,Z 826.638,A 0.000,B 0.000,C 90.000,E1 114.823} C_DIS
LIN {X -0.159,Y -368.739,Z 826.625,A 0.000,B 0.000,C 90.000,E1 112.461} C_DIS
LIN {X -0.169,Y -383.117,Z 826.612,A 0.000,B 0.000,C 90.000,E1 110.120} C_DIS
LIN {X -0.081,Y -398.934,Z 826.599,A 0.000,B 0.000,C 90.000,E1 107.819} C_DIS
LIN {X -0.226,Y -416.301,Z 826.587,A 0.000,B 0.000,C 90.000,E1 105.607} C_DIS
LIN {X -0.046,Y -435.330,Z 826.574,A 0.000,B 0.000,C 90.000,E1 103.411} C_DIS
LIN {X 0.004,Y -455.425,Z 826.563,A 0.000,B 0.000,C 90.000,E1 101.366} C_DIS
LIN {X -0.157,Y -468.178,Z 826.557,A 0.000,B 0.000,C 90.000,E1 100.197} C_DIS
LIN {X -0.177,Y -470.142,Z 826.555,A 0.000,B 0.000,C 90.000,E1 99.962} C_DIS
LIN {X -0.198,Y -471.634,Z 826.554,A 0.000,B 0.000,C 90.000,E1 99.726} C_DIS
LIN {X 0.044,Y -472.836,Z 826.552,A 0.000,B 0.000,C 90.000,E1 99.443} C_DIS
LIN {X -0.101,Y -473.714,Z 826.551,A 0.000,B 0.000,C 90.000,E1 99.208} C_DIS
LIN {X 0.087,Y -474.647,Z 826.548,A 0.000,B 0.000,C 90.000,E1 98.681} C_DIS
LIN {X 0.208,Y -474.601,Z 826.545,A 0.000,B 0.000,C 90.000,E1 98.163} C_DIS
LIN {X -0.134,Y -473.573,Z 826.543,A 0.000,B 0.000,C 90.000,E1 97.701} C_DIS
LIN {X 0.196,Y -472.647,Z 826.541,A 0.000,B 0.000,C 90.000,E1 97.409} C_DIS
LIN {X -0.005,Y -471.388,Z 826.540,A 0.000,B 0.000,C 90.000,E1 97.182} C_DIS
LIN {X 0.156,Y -453.680,Z 826.524,A 0.000,B 0.000,C 90.000,E1 94.359} C_DIS
LIN {X 0.038,Y -441.586,Z 826.513,A 0.000,B 0.000,C 90.000,E1 92.293} C_DIS
LIN {X 0.193,Y -432.276,Z 826.504,A 0.000,B 0.000,C 90.000,E1 90.688} C_DIS
LIN {X 0.173,Y -422.583,Z 826.495,A 0.000,B 0.000,C 90.000,E1 89.083} C_DIS
LIN {X 0.085,Y -411.181,Z 826.484,A 0.000,B 0.000,C 90.000,E1 87.192} C_DIS
LIN {X 0.138,Y -401.258,Z 826.475,A 0.000,B 0.000,C 90.000,E1 85.527} C_DIS
LIN {X 0.112,Y -386.526,Z 826.461,A 0.000,B 0.000,C 90.000,E1 82.996} C_DIS
LIN {X -0.146,Y -370.598,Z 826.445,A 0.000,B 0.000,C 90.000,E1 80.151} C_DIS
LIN {X -0.004,Y -355.494,Z 826.429,A 0.000,B 0.000,C 90.000,E1 77.173} C_DIS
LIN {X 0.080,Y -345.066,Z 826.417,A 0.000,B 0.000,C 90.000,E1 75.046} C_DIS
LIN {X 0.022,Y -334.743,Z 826.405,A 0.000,B 0.000,C 90.000,E1 72.906} C_DIS
LIN {X -0.095,Y -323.119,Z 826.391,A 0.000,B 0.000,C 90.000,E1 70.423} C_DIS
LIN {X -0.045,Y -310.412,Z 826.375,A 0.000,B 0.000,C 90.000,E1 67.539} C_DIS
LIN {X -0.111,Y -297.040,Z 826.357,A 0.000,B 0.000,C 90.000,E1 64.280} C_DIS
LIN {X 0.125,Y -288.075,Z 826.344,A 0.000,B 0.000,C 90.000,E1 61.897} C_DIS
LIN {X -0.038,Y -276.935,Z 826.327,A 0.000,B 0.000,C 90.000,E1 58.869} C_DIS
LIN {X -0.011,Y -265.264,Z 826.308,A 0.000,B 0.000,C 90.000,E1 55.388} C_DIS
LIN {X -0.034,Y -256.364,Z 826.292,A 0.000,B 0.000,C 90.000,E1 52.557} C_DIS
LIN {X 0.035,Y -245.671,Z 826.272,A 0.000,B 0.000,C 90.000,E1 48.933} C_DIS
LIN {X 0.058,Y -235.736,Z 826.251,A 0.000,B 0.000,C 90.000,E1 45.243} C_DIS
LIN {X -0.058,Y -226.594,Z 826.231,A 0.000,B 0.000,C 90.000,E1 41.515} C_DIS
LIN {X -0.076,Y -219.565,Z 826.214,A 0.000,B 0.000,C 90.000,E1 38.463} C_DIS
LIN {X 0.111,Y -212.823,Z 826.196,A 0.000,B 0.000,C 90.000,E1 35.311} C_DIS
LIN {X 0.054,Y -205.106,Z 826.174,A 0.000,B 0.000,C 90.000,E1 31.386} C_DIS
LIN {X -0.100,Y -199.600,Z 826.157,A 0.000,B 0.000,C 90.000,E1 28.231} C_DIS
LIN {X 0.047,Y -194.824,Z 826.139,A 0.000,B 0.000,C 90.000,E1 24.951} C_DIS
LIN {X 0.022,Y -189.936,Z 826.116,A 0.000,B 0.000,C 90.000,E1 20.865} C_DIS
LIN {X 0.009,Y -186.200,Z 826.093,A 0.000,B 0.000,C 90.000,E1 16.732} C_DIS
LIN {X 0.045,Y -183.257,Z 826.065,A 0.000,B 0.000,C 90.000,E1 11.715} C_DIS
LIN {X 0.013,Y -184.156,Z 825.969,A 0.000,B 0.000,C 90.000,E1 354.489} C_DIS
LIN {X 0.089,Y -187.484,Z 825.942,A 0.000,B 0.000,C 90.000,E1 349.454} C_DIS
LIN {X -0.007,Y -191.196,Z 825.919,A 0.000,B 0.000,C 90.000,E1 345.338} C_DIS
LIN {X 0.021,Y -195.829,Z 825.896,A 0.000,B 0.000,C 90.000,E1 341.221} C_DIS
LIN {X -0.056,Y -201.334,Z 825.873,A 0.000,B 0.000,C 90.000,E1 337.177} C_DIS
LIN {X 0.070,Y -207.663,Z 825.851,A 0.000,B 0.000,C 90.000,E1 333.127} C_DIS
LIN {X -0.056,Y -214.908,Z 825.829,A 0.000,B 0.000,C 90.000,E1 329.203} C_DIS
LIN {X -0.081,Y -221.319,Z 825.811,A 0.000,B 0.000,C 90.000,E1 326.087} C_DIS
LIN {X 0.069,Y -228.305,Z 825.794,A 0.000,B 0.000,C 90.000,E1 322.970} C_DIS
LIN {X -0.151,Y -235.946,Z 825.778,A 0.000,B 0.000,C 90.000,E1 319.989} C_DIS
LIN {X -0.081,Y -245.259,Z 825.759,A 0.000,B 0.000,C 90.000,E1 316.620} C_DIS
LIN {X 0.073,Y -255.533,Z 825.741,A 0.000,B 0.000,C 90.000,E1 313.299} C_DIS
LIN {X 0.023,Y -266.525,Z 825.723,A 0.000,B 0.000,C 90.000,E1 310.092} C_DIS
LIN {X 0.087,Y -279.820,Z 825.703,A 0.000,B 0.000,C 90.000,E1 306.583} C_DIS
LIN {X 0.161,Y -292.955,Z 825.686,A 0.000,B 0.000,C 90.000,E1 303.499} C_DIS
LIN {X 0.007,Y -309.100,Z 825.668,A 0.000,B 0.000,C 90.000,E1 300.207} C_DIS
LIN {X -0.118,Y -323.501,Z 825.653,A 0.000,B 0.000,C 90.000,E1 297.641} C_DIS
LIN {X -0.008,Y -337.223,Z 825.641,A 0.000,B 0.000,C 90.000,E1 295.412} C_DIS
LIN {X -0.051,Y -351.841,Z 825.629,A 0.000,B 0.000,C 90.000,E1 293.259} C_DIS
LIN {X 0.022,Y -370.136,Z 825.616,A 0.000,B 0.000,C 90.000,E1 290.844} C_DIS
LIN {X 0.030,Y -395.352,Z 825.600,A 0.000,B 0.000,C 90.000,E1 287.946} C_DIS
LIN {X 0.015,Y -408.168,Z 825.592,A 0.000,B 0.000,C 90.000,E1 286.567} C_DIS
LIN {X -0.060,Y -420.645,Z 825.585,A 0.000,B 0.000,C 90.000,E1 285.245} C_DIS
LIN {X 0.136,Y -432.928,Z 825.577,A 0.000,B 0.000,C 90.000,E1 283.883} C_DIS
LIN {X 0.053,Y -442.675,Z 825.571,A 0.000,B 0.000,C 90.000,E1 282.827} C_DIS
LIN {X 0.086,Y -451.808,Z 825.565,A 0.000,B 0.000,C 90.000,E1 281.771} C_DIS
LIN {X 0.139,Y -460.453,Z 825.560,A 0.000,B 0.000,C 90.000,E1 280.725} C_DIS
LIN {X -0.079,Y -468.362,Z 825.554,A 0.000,B 0.000,C 90.000,E1 279.726} C_DIS
LIN {X -0.157,Y -473.791,Z 825.550,A 0.000,B 0.000,C 90.000,E1 278.973} C_DIS
LIN {X -0.182,Y -478.632,Z 825.546,A 0.000,B 0.000,C 90.000,E1 278.219} C_DIS
LIN {X -0.170,Y -482.850,Z 825.541,A 0.000,B 0.000,C 90.000,E1 277.466} C_DIS
LIN {X -0.176,Y -486.388,Z 825.537,A 0.000,B 0.000,C 90.000,E1 276.720} C_DIS
LIN {X -0.097,Y -489.181,Z 825.533,A 0.000,B 0.000,C 90.000,E1 275.967} C_DIS
LIN {X 0.062,Y -490.572,Z 825.530,A 0.000,B 0.000,C 90.000,E1 275.454} C_DIS
LIN {X -0.207,Y -491.625,Z 825.528,A 0.000,B 0.000,C 90.000,E1 274.992} C_DIS
LIN {X 0.018,Y -492.370,Z 825.525,A 0.000,B 0.000,C 90.000,E1 274.473} C_DIS
LIN {X 0.248,Y -492.692,Z 825.522,A 0.000,B 0.000,C 90.000,E1 273.955} C_DIS
LIN {X -0.043,Y -492.637,Z 825.519,A 0.000,B 0.000,C 90.000,E1 273.498} C_DIS
LIN {X 0.190,Y -492.204,Z 825.517,A 0.000,B 0.000,C 90.000,E1 272.980} C_DIS
LIN {X -0.095,Y -491.354,Z 825.514,A 0.000,B 0.000,C 90.000,E1 272.522} C_DIS
LIN {X 0.111,Y -490.129,Z 825.511,A 0.000,B 0.000,C 90.000,E1 272.007} C_DIS
LIN {X -0.162,Y -488.428,Z 825.508,A 0.000,B 0.000,C 90.000,E1 271.547} C_DIS
LIN {X 0.032,Y -486.261,Z 825.506,A 0.000,B 0.000,C 90.000,E1 271.031} C_DIS
LIN {X 0.216,Y -483.491,Z 825.503,A 0.000,B 0.000,C 90.000,E1 270.516} C_DIS
LIN {X -0.102,Y -480.094,Z 825.500,A 0.000,B 0.000,C 90.000,E1 270.057} C_DIS
LIN {X 0.044,Y -475.968,Z 825.497,A 0.000,B 0.000,C 90.000,E1 269.542} C_DIS
LIN {X 0.166,Y -470.891,Z 825.495,A 0.000,B 0.000,C 90.000,E1 269.026} C_DIS
LIN {X 0.082,Y -468.104,Z 825.493,A 0.000,B 0.000,C 90.000,E1 268.797} C_DIS
LIN {X 0.173,Y -461.956,Z 825.491,A 0.000,B 0.000,C 90.000,E1 268.339} C_DIS
LIN {X -0.129,Y -455.303,Z 825.489,A 0.000,B 0.000,C 90.000,E1 267.993} C_DIS
LIN {X 0.115,Y -447.961,Z 825.487,A 0.000,B 0.000,C 90.000,E1 267.650} C_DIS
LIN {X -0.010,Y -440.279,Z 825.486,A 0.000,B 0.000,C 90.000,E1 267.421} C_DIS
LIN {X -0.094,Y -431.941,Z 825.485,A 0.000,B 0.000,C 90.000,E1 267.249} C_DIS
LIN {X -0.131,Y -421.863,Z 825.484,A 0.000,B 0.000,C 90.000,E1 267.135} C_DIS
LIN {X 0.191,Y -417.695,Z 825.484,A 0.000,B 0.000,C 90.000,E1 267.078} C_DIS
LIN {X 0.062,Y -181.002,Z 825.484,A 0.000,B 0.000,C 90.000,E1 267.078} C_DIS
LIN {X 0.074,Y -180.906,Z 825.474,A 0.000,B 0.000,C 90.000,E1 265.355} C_DIS
LIN {X -0.032,Y -180.693,Z 825.470,A 0.000,B 0.000,C 90.000,E1 264.546} C_DIS
LIN {X 0.046,Y -178.778,Z 825.441,A 0.000,B 0.000,C 90.000,E1 259.454} C_DIS
LIN {X -0.052,Y -175.825,Z 825.413,A 0.000,B 0.000,C 90.000,E1 254.393} C_DIS
LIN {X -0.051,Y -172.012,Z 825.385,A 0.000,B 0.000,C 90.000,E1 249.263} C_DIS
LIN {X -0.074,Y -171.432,Z 825.380,A 0.000,B 0.000,C 90.000,E1 248.411} C_DIS
LIN {X -0.019,Y -167.668,Z 825.356,A 0.000,B 0.000,C 90.000,E1 244.076} C_DIS
LIN {X -0.079,Y -166.341,Z 825.346,A 0.000,B 0.000,C 90.000,E1 242.359} C_DIS
LIN {X -0.086,Y -163.078,Z 825.327,A 0.000,B 0.000,C 90.000,E1 238.869} C_DIS
LIN {X -0.035,Y -161.018,Z 825.312,A 0.000,B 0.000,C 90.000,E1 236.215} C_DIS
LIN {X -0.050,Y -157.760,Z 825.293,A 0.000,B 0.000,C 90.000,E1 232.683} C_DIS
LIN {X 0.013,Y -155.799,Z 825.278,A 0.000,B 0.000,C 90.000,E1 229.989} C_DIS
LIN {X 0.067,Y -152.051,Z 825.253,A 0.000,B 0.000,C 90.000,E1 225.486} C_DIS
LIN {X 0.084,Y -150.300,Z 825.238,A 0.000,B 0.000,C 90.000,E1 222.771} C_DIS
LIN {X 0.009,Y -147.046,Z 825.213,A 0.000,B 0.000,C 90.000,E1 218.257} C_DIS
LIN {X 0.003,Y -145.625,Z 825.197,A 0.000,B 0.000,C 90.000,E1 215.518} C_DIS
LIN {X 0.001,Y -143.009,Z 825.172,A 0.000,B 0.000,C 90.000,E1 210.924} C_DIS
LIN {X -0.068,Y -141.636,Z 825.151,A 0.000,B 0.000,C 90.000,E1 207.257} C_DIS
LIN {X -0.017,Y -139.437,Z 825.115,A 0.000,B 0.000,C 90.000,E1 200.737} C_DIS
LIN {X 0.037,Y -139.169,Z 825.105,A 0.000,B 0.000,C 90.000,E1 198.852} C_DIS
LIN {X -0.066,Y -138.317,Z 825.053,A 0.000,B 0.000,C 90.000,E1 189.557} C_DIS
LIN {X -0.057,Y -139.474,Z 825.006,A 0.000,B 0.000,C 90.000,E1 181.146} C_DIS
LIN {X 0.024,Y -141.051,Z 824.975,A 0.000,B 0.000,C 90.000,E1 175.527} C_DIS
LIN {X -0.022,Y -142.422,Z 824.960,A 0.000,B 0.000,C 90.000,E1 172.761} C_DIS
LIN {X 0.038,Y -144.658,Z 824.934,A 0.000,B 0.000,C 90.000,E1 168.117} C_DIS
LIN {X 0.022,Y -147.241,Z 824.914,A 0.000,B 0.000,C 90.000,E1 164.448} C_DIS
LIN {X 0.041,Y -150.557,Z 824.888,A 0.000,B 0.000,C 90.000,E1 159.880} C_DIS
LIN {X -0.020,Y -154.025,Z 824.868,A 0.000,B 0.000,C 90.000,E1 156.282} C_DIS
LIN {X 0.048,Y -157.440,Z 824.848,A 0.000,B 0.000,C 90.000,E1 152.666} C_DIS
LIN {X -0.002,Y -161.656,Z 824.828,A 0.000,B 0.000,C 90.000,E1 149.125} C_DIS
LIN {X 0.015,Y -165.851,Z 824.809,A 0.000,B 0.000,C 90.000,E1 145.595} C_DIS
LIN {X 0.007,Y -170.826,Z 824.789,A 0.000,B 0.000,C 90.000,E1 142.110} C_DIS
LIN {X -0.078,Y -175.695,Z 824.770,A 0.000,B 0.000,C 90.000,E1 138.690} C_DIS
LIN {X 0.046,Y -181.308,Z 824.751,A 0.000,B 0.000,C 90.000,E1 135.243} C_DIS
LIN {X -0.082,Y -186.789,Z 824.733,A 0.000,B 0.000,C 90.000,E1 131.919} C_DIS
LIN {X -0.012,Y -191.382,Z 824.719,A 0.000,B 0.000,C 90.000,E1 129.402} C_DIS
LIN {X 0.006,Y -192.801,Z 824.714,A 0.000,B 0.000,C 90.000,E1 128.543} C_DIS
LIN {X -0.045,Y -293.702,Z 824.714,A 0.000,B 0.000,C 90.000,E1 128.543} C_DIS
LIN {X -0.022,Y -295.264,Z 824.714,A 0.000,B 0.000,C 90.000,E1 128.508} C_DIS
LIN {X 0.068,Y -299.226,Z 824.713,A 0.000,B 0.000,C 90.000,E1 128.302} C_DIS
LIN {X 0.161,Y -301.530,Z 824.712,A 0.000,B 0.000,C 90.000,E1 128.096} C_DIS
LIN {X 0.109,Y -304.699,Z 824.710,A 0.000,B 0.000,C 90.000,E1 127.729} C_DIS
LIN {X -0.081,Y -306.645,Z 824.708,A 0.000,B 0.000,C 90.000,E1 127.443} C_DIS
LIN {X 0.160,Y -308.161,Z 824.706,A 0.000,B 0.000,C 90.000,E1 127.076} C_DIS
LIN {X -0.059,Y -309.374,Z 824.704,A 0.000,B 0.000,C 90.000,E1 126.790} C_DIS
LIN {X 0.027,Y -320.434,Z 824.685,A 0.000,B 0.000,C 90.000,E1 123.214} C_DIS
LIN {X 0.151,Y -330.833,Z 824.669,A 0.000,B 0.000,C 90.000,E1 120.335} C_DIS
LIN {X -0.052,Y -342.585,Z 824.653,A 0.000,B 0.000,C 90.000,E1 117.564} C_DIS
LIN {X -0.103,Y -355.789,Z 824.638,A 0.000,B 0.000,C 90.000,E1 114.823} C_DIS
LIN {X 0.040,Y -368.844,Z 824.625,A 0.000,B 0.000,C 90.000,E1 112.408} C_DIS
LIN {X 0.046,Y -383.235,Z 824.612,A 0.000,B 0.000,C 90.000,E1 110.066} C_DIS
LIN {X 0.150,Y -399.064,Z 824.599,A 0.000,B 0.000,C 90.000,E1 107.764} C_DIS
LIN {X 0.023,Y -416.447,Z 824.586,A 0.000,B 0.000,C 90.000,E1 105.552} C_DIS
LIN {X 0.223,Y -435.491,Z 824.574,A 0.000,B 0.000,C 90.000,E1 103.355} C_DIS
LIN {X -0.146,Y -455.591,Z 824.563,A 0.000,B 0.000,C 90.000,E1 101.366} C_DIS
LIN {X 0.157,Y -468.322,Z 824.556,A 0.000,B 0.000,C 90.000,E1 100.141} C_DIS
LIN {X 0.128,Y -470.260,Z 824.555,A 0.000,B 0.000,C 90.000,E1 99.905} C_DIS
LIN {X 0.096,Y -471.733,Z 824.554,A 0.000,B 0.000,C 90.000,E1 99.670} C_DIS
LIN {X 0.195,Y -473.765,Z 824.551,A 0.000,B 0.000,C 90.000,E1 99.151} C_DIS
LIN {X -0.091,Y -474.662,Z 824.548,A 0.000,B 0.000,C 90.000,E1 98.681} C_DIS
LIN {X 0.030,Y -474.580,Z 824.545,A 0.000,B 0.000,C 90.000,E1 98.163} C_DIS
LIN {X 0.158,Y -473.513,Z 824.543,A 0.000,B 0.000,C 90.000,E1 97.644} C_DIS
LIN {X 0.018,Y -472.563,Z 824.541,A 0.000,B 0.000,C 90.000,E1 97.409} C_DIS
LIN {X -0.181,Y -471.277,Z 824.540,A 0.000,B 0.000,C 90.000,E1 97.182} C_DIS
LIN {X -0.017,Y -453.586,Z 824.524,A 0.000,B 0.000,C 90.000,E1 94.359} C_DIS
LIN {X -0.133,Y -441.491,Z 824.513,A 0.000,B 0.000,C 90.000,E1 92.293} C_DIS
LIN {X 0.025,Y -432.196,Z 824.504,A 0.000,B 0.000,C 90.000,E1 90.688} C_DIS
LIN {X 0.007,Y -422.502,Z 824.495,A 0.000,B 0.000,C 90.000,E1 89.083} C_DIS
LIN {X -0.169,Y -412.739,Z 824.486,A 0.000,B 0.000,C 90.000,E1 87.478} C_DIS
LIN {X -0.023,Y -401.175,Z 824.475,A 0.000,B 0.000,C 90.000,E1 85.527} C_DIS
LIN {X -0.045,Y -386.444,Z 824.461,A 0.000,B 0.000,C 90.000,E1 82.996} C_DIS
LIN {X 0.065,Y -370.520,Z 824.445,A 0.000,B 0.000,C 90.000,E1 80.095} C_DIS
LIN {X -0.153,Y -355.432,Z 824.429,A 0.000,B 0.000,C 90.000,E1 77.173} C_DIS
LIN {X -0.066,Y -345.013,Z 824.417,A 0.000,B 0.000,C 90.000,E1 75.046} C_DIS
LIN {X -0.133,Y -333.253,Z 824.403,A 0.000,B 0.000,C 90.000,E1 72.598} C_DIS
LIN {X 0.026,Y -321.675,Z 824.389,A 0.000,B 0.000,C 90.000,E1 70.061} C_DIS
LIN {X 0.022,Y -309.076,Z 824.373,A 0.000,B 0.000,C 90.000,E1 67.177} C_DIS
LIN {X 0.034,Y -295.820,Z 824.355,A 0.000,B 0.000,C 90.000,E1 63.896} C_DIS
LIN {X -0.010,Y -286.927,Z 824.342,A 0.000,B 0.000,C 90.000,E1 61.563} C_DIS
LIN {X 0.036,Y -275.917,Z 824.325,A 0.000,B 0.000,C 90.000,E1 58.486} C_DIS
LIN {X -0.049,Y -264.383,Z 824.306,A 0.000,B 0.000,C 90.000,E1 55.022} C_DIS
LIN {X -0.128,Y -256.636,Z 824.292,A 0.000,B 0.000,C 90.000,E1 52.557} C_DIS
LIN {X -0.046,Y -245.958,Z 824.272,A 0.000,B 0.000,C 90.000,E1 48.933} C_DIS
LIN {X -0.011,Y -236.012,Z 824.251,A 0.000,B 0.000,C 90.000,E1 45.243} C_DIS
LIN {X 0.055,Y -226.895,Z 824.230,A 0.000,B 0.000,C 90.000,E1 41.472} C_DIS
LIN {X -0.124,Y -219.893,Z 824.214,A 0.000,B 0.000,C 90.000,E1 38.463} C_DIS
LIN {X 0.071,Y -213.118,Z 824.196,A 0.000,B 0.000,C 90.000,E1 35.311} C_DIS
LIN {X 0.025,Y -205.414,Z 824.174,A 0.000,B 0.000,C 90.000,E1 31.386} C_DIS
LIN {X 0.055,Y -199.899,Z 824.157,A 0.000,B 0.000,C 90.000,E1 28.180} C_DIS
LIN {X 0.033,Y -195.138,Z 824.139,A 0.000,B 0.000,C 90.000,E1 24.951} C_DIS
LIN {X 0.019,Y -190.248,Z 824.116,A 0.000,B 0.000,C 90.000,E1 20.865} C_DIS
LIN {X 0.015,Y -186.491,Z 824.093,A 0.000,B 0.000,C 90.000,E1 16.732} C_DIS
LIN {X 0.062,Y -183.568,Z 824.065,A 0.000,B 0.000,C 90.000,E1 11.715} C_DIS
LIN {X 0.024,Y -184.434,Z 823.969,A 0.000,B 0.000,C 90.000,E1 354.489} C_DIS
LIN {X -0.075,Y -187.734,Z 823.942,A 0.000,B 0.000,C 90.000,E1 349.511} C_DIS
LIN {X 0.022,Y -191.429,Z 823.919,A 0.000,B 0.000,C 90.000,E1 345.338} C_DIS
LIN {X 0.058,Y -196.042,Z 823.896,A 0.000,B 0.000,C 90.000,E1 341.221} C_DIS
LIN {X -0.011,Y -201.524,Z 823.873,A 0.000,B 0.000,C 90.000,E1 337.177} C_DIS
LIN {X -0.063,Y -207.861,Z 823.851,A 0.000,B 0.000,C 90.000,E1 333.179} C_DIS
LIN {X 0.005,Y -215.099,Z 823.829,A 0.000,B 0.000,C 90.000,E1 329.203} C_DIS
LIN {X -0.014,Y -221.534,Z 823.812,A 0.000,B 0.000,C 90.000,E1 326.087} C_DIS
LIN {X -0.111,Y -230.327,Z 823.790,A 0.000,B 0.000,C 90.000,E1 322.271} C_DIS
LIN {X -0.012,Y -239.161,Z 823.771,A 0.000,B 0.000,C 90.000,E1 318.852} C_DIS
LIN {X 0.147,Y -248.701,Z 823.753,A 0.000,B 0.000,C 90.000,E1 315.486} C_DIS
LIN {X 0.066,Y -259.220,Z 823.735,A 0.000,B 0.000,C 90.000,E1 312.243} C_DIS
LIN {X -0.047,Y -270.488,Z 823.717,A 0.000,B 0.000,C 90.000,E1 309.072} C_DIS
LIN {X 0.029,Y -282.643,Z 823.700,A 0.000,B 0.000,C 90.000,E1 305.931} C_DIS
LIN {X 0.012,Y -297.566,Z 823.681,A 0.000,B 0.000,C 90.000,E1 302.546} C_DIS
LIN {X -0.055,Y -312.493,Z 823.664,A 0.000,B 0.000,C 90.000,E1 299.589} C_DIS
LIN {X -0.053,Y -325.314,Z 823.652,A 0.000,B 0.000,C 90.000,E1 297.334} C_DIS
LIN {X -0.088,Y -343.148,Z 823.636,A 0.000,B 0.000,C 90.000,E1 294.515} C_DIS
LIN {X 0.187,Y -358.273,Z 823.624,A 0.000,B 0.000,C 90.000,E1 292.333} C_DIS
LIN {X -0.044,Y -377.131,Z 823.611,A 0.000,B 0.000,C 90.000,E1 289.993} C_DIS
LIN {X -0.098,Y -394.854,Z 823.600,A 0.000,B 0.000,C 90.000,E1 288.000} C_DIS
LIN {X 0.154,Y -410.159,Z 823.591,A 0.000,B 0.000,C 90.000,E1 286.315} C_DIS
LIN {X -0.044,Y -422.605,Z 823.583,A 0.000,B 0.000,C 90.000,E1 285.009} C_DIS
LIN {X 0.067,Y -434.936,Z 823.576,A 0.000,B 0.000,C 90.000,E1 283.647} C_DIS
LIN {X 0.006,Y -444.619,Z 823.570,A 0.000,B 0.000,C 90.000,E1 282.591} C_DIS
LIN {X 0.060,Y -453.668,Z 823.564,A 0.000,B 0.000,C 90.000,E1 281.535} C_DIS
LIN {X 0.134,Y -462.145,Z 823.558,A 0.000,B 0.000,C 90.000,E1 280.489} C_DIS
LIN {X -0.146,Y -469.887,Z 823.553,A 0.000,B 0.000,C 90.000,E1 279.500} C_DIS
LIN {X -0.202,Y -475.168,Z 823.548,A 0.000,B 0.000,C 90.000,E1 278.746} C_DIS
LIN {X -0.216,Y -479.838,Z 823.544,A 0.000,B 0.000,C 90.000,E1 277.992} C_DIS
LIN {X -0.187,Y -483.845,Z 823.540,A 0.000,B 0.000,C 90.000,E1 277.239} C_DIS
LIN {X -0.129,Y -487.202,Z 823.536,A 0.000,B 0.000,C 90.000,E1 276.486} C_DIS
LIN {X 0.070,Y -488.999,Z 823.533,A 0.000,B 0.000,C 90.000,E1 275.967} C_DIS
LIN {X -0.260,Y -490.456,Z 823.530,A 0.000,B 0.000,C 90.000,E1 275.511} C_DIS
LIN {X -0.041,Y -491.567,Z 823.528,A 0.000,B 0.000,C 90.000,E1 274.992} C_DIS
LIN {X 0.184,Y -492.297,Z 823.525,A 0.000,B 0.000,C 90.000,E1 274.473} C_DIS
LIN {X -0.078,Y -492.650,Z 823.522,A 0.000,B 0.000,C 90.000,E1 274.012} C_DIS
LIN {X 0.122,Y -492.654,Z 823.520,A 0.000,B 0.000,C 90.000,E1 273.498} C_DIS
LIN {X -0.137,Y -492.231,Z 823.517,A 0.000,B 0.000,C 90.000,E1 273.037} C_DIS
LIN {X 0.069,Y -491.441,Z 823.514,A 0.000,B 0.000,C 90.000,E1 272.522} C_DIS
LIN {X -0.216,Y -490.234,Z 823.511,A 0.000,B 0.000,C 90.000,E1 272.064} C_DIS
LIN {X 0.002,Y -488.595,Z 823.509,A 0.000,B 0.000,C 90.000,E1 271.547} C_DIS
LIN {X 0.195,Y -486.449,Z 823.506,A 0.000,B 0.000,C 90.000,E1 271.031} C_DIS
LIN {X -0.104,Y -483.739,Z 823.503,A 0.000,B 0.000,C 90.000,E1 270.573} C_DIS
LIN {X 0.062,Y -480.409,Z 823.500,A 0.000,B 0.000,C 90.000,E1 270.057} C_DIS
LIN {X 0.209,Y -476.346,Z 823.498,A 0.000,B 0.000,C 90.000,E1 269.542} C_DIS
LIN {X -0.141,Y -471.367,Z 823.495,A 0.000,B 0.000,C 90.000,E1 269.083} C_DIS
LIN {X 0.110,Y -465.493,Z 823.492,A 0.000,B 0.000,C 90.000,E1 268.568} C_DIS
LIN {X -0.212,Y -462.480,Z 823.491,A 0.000,B 0.000,C 90.000,E1 268.396} C_DIS
LIN {X -0.088,Y -455.828,Z 823.489,A 0.000,B 0.000,C 90.000,E1 267.993} C_DIS
LIN {X 0.121,Y -448.564,Z 823.487,A 0.000,B 0.000,C 90.000,E1 267.650} C_DIS
LIN {X -0.044,Y -440.820,Z 823.486,A 0.000,B 0.000,C 90.000,E1 267.421} C_DIS
LIN {X -0.153,Y -432.717,Z 823.485,A 0.000,B 0.000,C 90.000,E1 267.249} C_DIS
LIN {X -0.207,Y -423.321,Z 823.484,A 0.000,B 0.000,C 90.000,E1 267.135} C_DIS
LIN {X 0.058,Y -419.228,Z 823.484,A 0.000,B 0.000,C 90.000,E1 267.078} C_DIS
LIN {X 0.002,Y -181.000,Z 823.484,A 0.000,B 0.000,C 90.000,E1 267.078} C_DIS
LIN {X 0.029,Y -180.906,Z 823.474,A 0.000,B 0.000,C 90.000,E1 265.355} C_DIS
LIN {X -0.077,Y -180.686,Z 823.470,A 0.000,B 0.000,C 90.000,E1 264.546} C_DIS
LIN {X 0.000,Y -178.769,Z 823.441,A 0.000,B 0.000,C 90.000,E1 259.454} C_DIS
LIN {X 0.073,Y -175.816,Z 823.413,A 0.000,B 0.000,C 90.000,E1 254.338} C_DIS
LIN {X 0.066,Y -172.003,Z 823.385,A 0.000,B 0.000,C 90.000,E1 249.209} C_DIS
LIN {X 0.041,Y -171.420,Z 823.380,A 0.000,B 0.000,C 90.000,E1 248.358} C_DIS
LIN {X 0.087,Y -167.658,Z 823.356,A 0.000,B 0.000,C 90.000,E1 244.024} C_DIS
LIN {X 0.025,Y -166.325,Z 823.346,A 0.000,B 0.000,C 90.000,E1 242.308} C_DIS
LIN {X 0.011,Y -163.066,Z 823.327,A 0.000,B 0.000,C 90.000,E1 238.820} C_DIS
LIN {X -0.077,Y -161.003,Z 823.312,A 0.000,B 0.000,C 90.000,E1 236.215} C_DIS
LIN {X 0.033,Y -157.748,Z 823.292,A 0.000,B 0.000,C 90.000,E1 232.637} C_DIS
LIN {X -0.029,Y -155.787,Z 823.278,A 0.000,B 0.000,C 90.000,E1 229.989} C_DIS
LIN {X 0.026,Y -152.040,Z 823.253,A 0.000,B 0.000,C 90.000,E1 225.486} C_DIS
LIN {X 0.044,Y -150.289,Z 823.238,A 0.000,B 0.000,C 90.000,E1 222.771} C_DIS
LIN {X -0.030,Y -147.037,Z 823.212,A 0.000,B 0.000,C 90.000,E1 218.257} C_DIS
LIN {X -0.037,Y -145.618,Z 823.197,A 0.000,B 0.000,C 90.000,E1 215.518} C_DIS
LIN {X -0.038,Y -143.002,Z 823.172,A 0.000,B 0.000,C 90.000,E1 210.924} C_DIS
LIN {X 0.019,Y -141.628,Z 823.151,A 0.000,B 0.000,C 90.000,E1 207.206} C_DIS
LIN {X -0.056,Y -139.435,Z 823.115,A 0.000,B 0.000,C 90.000,E1 200.737} C_DIS
LIN {X -0.002,Y -139.166,Z 823.105,A 0.000,B 0.000,C 90.000,E1 198.852} C_DIS
LIN {X 0.032,Y -138.316,Z 823.053,A 0.000,B 0.000,C 90.000,E1 189.500} C_DIS
LIN {X 0.043,Y -139.476,Z 823.006,A 0.000,B 0.000,C 90.000,E1 181.088} C_DIS
LIN {X -0.016,Y -141.058,Z 822.975,A 0.000,B 0.000,C 90.000,E1 175.527} C_DIS
LIN {X -0.062,Y -142.430,Z 822.960,A 0.000,B 0.000,C 90.000,E1 172.761} C_DIS
LIN {X -0.002,Y -144.667,Z 822.934,A 0.000,B 0.000,C 90.000,E1 168.117} C_DIS
LIN {X -0.018,Y -147.253,Z 822.914,A 0.000,B 0.000,C 90.000,E1 164.448} C_DIS
LIN {X 0.000,Y -150.570,Z 822.888,A 0.000,B 0.000,C 90.000,E1 159.880} C_DIS
LIN {X 0.079,Y -154.040,Z 822.868,A 0.000,B 0.000,C 90.000,E1 156.230} C_DIS
LIN {X 0.006,Y -157.456,Z 822.848,A 0.000,B 0.000,C 90.000,E1 152.666} C_DIS
LIN {X -0.045,Y -161.676,Z 822.828,A 0.000,B 0.000,C 90.000,E1 149.125} C_DIS
LIN {X -0.028,Y -165.870,Z 822.809,A 0.000,B 0.000,C 90.000,E1 145.595} C_DIS
LIN {X -0.038,Y -170.849,Z 822.789,A 0.000,B 0.000,C 90.000,E1 142.110} C_DIS
LIN {X 0.010,Y -175.718,Z 822.770,A 0.000,B 0.000,C 90.000,E1 138.647} C_DIS
LIN {X 0.000,Y -181.329,Z 822.751,A 0.000,B 0.000,C 90.000,E1 135.243} C_DIS
LIN {X -0.004,Y -186.815,Z 822.733,A 0.000,B 0.000,C 90.000,E1 131.881} C_DIS
LIN {X -0.058,Y -191.405,Z 822.719,A 0.000,B 0.000,C 90.000,E1 129.402} C_DIS
LIN {X 0.028,Y -192.790,Z 822.714,A 0.000,B 0.000,C 90.000,E1 128.543} C_DIS
LIN {X 0.008,Y -293.475,Z 822.714,A 0.000,B 0.000,C 90.000,E1 128.543} C_DIS
LIN {X 0.136,Y -295.931,Z 822.714,A 0.000,B 0.000,C 90.000,E1 128.463} C_DIS
LIN {X -0.006,Y -299.498,Z 822.713,A 0.000,B 0.000,C 90.000,E1 128.302} C_DIS
LIN {X 0.086,Y -301.714,Z 822.712,A 0.000,B 0.000,C 90.000,E1 128.096} C_DIS
LIN {X 0.034,Y -304.807,Z 822.710,A 0.000,B 0.000,C 90.000,E1 127.729} C_DIS
LIN {X 0.059,Y -306.747,Z 822.708,A 0.000,B 0.000,C 90.000,E1 127.397} C_DIS
LIN {X 0.025,Y -308.255,Z 822.706,A 0.000,B 0.000,C 90.000,E1 127.076} C_DIS
LIN {X 0.020,Y -310.397,Z 822.702,A 0.000,B 0.000,C 90.000,E1 126.423} C_DIS
LIN {X 0.158,Y -320.496,Z 822.684,A 0.000,B 0.000,C 90.000,E1 123.166} C_DIS
LIN {X 0.009,Y -330.906,Z 822.669,A 0.000,B 0.000,C 90.000,E1 120.335} C_DIS
LIN {X 0.107,Y -342.671,Z 822.653,A 0.000,B 0.000,C 90.000,E1 117.513} C_DIS
LIN {X 0.073,Y -355.887,Z 822.638,A 0.000,B 0.000,C 90.000,E1 114.771} C_DIS
LIN {X 0.030,Y -368.955,Z 822.624,A 0.000,B 0.000,C 90.000,E1 112.386} C_DIS
LIN {X -0.107,Y -383.359,Z 822.611,A 0.000,B 0.000,C 90.000,E1 110.066} C_DIS
LIN {X -0.006,Y -399.203,Z 822.599,A 0.000,B 0.000,C 90.000,E1 107.764} C_DIS
LIN {X -0.136,Y -416.602,Z 822.586,A 0.000,B 0.000,C 90.000,E1 105.552} C_DIS
LIN {X 0.061,Y -435.661,Z 822.574,A 0.000,B 0.000,C 90.000,E1 103.355} C_DIS
LIN {X 0.235,Y -455.767,Z 822.563,A 0.000,B 0.000,C 90.000,E1 101.299} C_DIS
LIN {X 0.005,Y -468.468,Z 822.556,A 0.000,B 0.000,C 90.000,E1 100.141} C_DIS
LIN {X -0.041,Y -470.381,Z 822.555,A 0.000,B 0.000,C 90.000,E1 99.905} C_DIS
LIN {X -0.088,Y -471.835,Z 822.554,A 0.000,B 0.000,C 90.000,E1 99.670} C_DIS
LIN {X 0.012,Y -473.816,Z 822.551,A 0.000,B 0.000,C 90.000,E1 99.151} C_DIS
LIN {X 0.194,Y -474.673,Z 822.548,A 0.000,B 0.000,C 90.000,E1 98.624} C_DIS
LIN {X -0.153,Y -474.554,Z 822.545,A 0.000,B 0.000,C 90.000,E1 98.163} C_DIS
LIN {X -0.024,Y -473.448,Z 822.542,A 0.000,B 0.000,C 90.000,E1 97.644} C_DIS
LIN {X -0.164,Y -472.474,Z 822.541,A 0.000,B 0.000,C 90.000,E1 97.409} C_DIS
LIN {X 0.105,Y -471.159,Z 822.540,A 0.000,B 0.000,C 90.000,E1 97.125} C_DIS
LIN {X -0.195,Y -453.488,Z 822.524,A 0.000,B 0.000,C 90.000,E1 94.359} C_DIS
LIN {X 0.133,Y -441.388,Z 822.513,A 0.000,B 0.000,C 90.000,E1 92.236} C_DIS
LIN {X 0.129,Y -433.687,Z 822.505,A 0.000,B 0.000,C 90.000,E1 90.917} C_DIS
LIN {X 0.135,Y -424.054,Z 822.496,A 0.000,B 0.000,C 90.000,E1 89.312} C_DIS
LIN {X -0.017,Y -414.303,Z 822.487,A 0.000,B 0.000,C 90.000,E1 87.707} C_DIS
LIN {X 0.072,Y -404.414,Z 822.478,A 0.000,B 0.000,C 90.000,E1 86.045} C_DIS
LIN {X 0.120,Y -391.233,Z 822.466,A 0.000,B 0.000,C 90.000,E1 83.799} C_DIS
LIN {X -0.088,Y -378.294,Z 822.453,A 0.000,B 0.000,C 90.000,E1 81.546} C_DIS
LIN {X -0.124,Y -364.259,Z 822.438,A 0.000,B 0.000,C 90.000,E1 78.926} C_DIS
LIN {X 0.021,Y -352.387,Z 822.425,A 0.000,B 0.000,C 90.000,E1 76.520} C_DIS
LIN {X 0.041,Y -342.003,Z 822.413,A 0.000,B 0.000,C 90.000,E1 74.393} C_DIS
LIN {X 0.017,Y -331.738,Z 822.401,A 0.000,B 0.000,C 90.000,E1 72.236} C_DIS
LIN {X 0.134,Y -320.251,Z 822.387,A 0.000,B 0.000,C 90.000,E1 69.699} C_DIS
LIN {X 0.116,Y -306.389,Z 822.370,A 0.000,B 0.000,C 90.000,E1 66.485} C_DIS
LIN {X 0.043,Y -293.366,Z 822.351,A 0.000,B 0.000,C 90.000,E1 63.204} C_DIS
LIN {X -0.117,Y -282.108,Z 822.334,A 0.000,B 0.000,C 90.000,E1 60.205} C_DIS
LIN {X -0.012,Y -271.396,Z 822.317,A 0.000,B 0.000,C 90.000,E1 57.089} C_DIS
LIN {X 0.035,Y -262.406,Z 822.302,A 0.000,B 0.000,C 90.000,E1 54.276} C_DIS
LIN {X 0.056,Y -254.716,Z 822.288,A 0.000,B 0.000,C 90.000,E1 51.778} C_DIS
LIN {X -0.136,Y -246.237,Z 822.272,A 0.000,B 0.000,C 90.000,E1 48.933} C_DIS
LIN {X -0.089,Y -236.284,Z 822.251,A 0.000,B 0.000,C 90.000,E1 45.243} C_DIS
LIN {X -0.012,Y -227.185,Z 822.230,A 0.000,B 0.000,C 90.000,E1 41.472} C_DIS
LIN {X 0.126,Y -220.200,Z 822.213,A 0.000,B 0.000,C 90.000,E1 38.382} C_DIS
LIN {X 0.023,Y -213.407,Z 822.196,A 0.000,B 0.000,C 90.000,E1 35.311} C_DIS
LIN {X -0.013,Y -205.713,Z 822.174,A 0.000,B 0.000,C 90.000,E1 31.386} C_DIS
LIN {X 0.025,Y -200.186,Z 822.157,A 0.000,B 0.000,C 90.000,E1 28.180} C_DIS
LIN {X 0.012,Y -195.430,Z 822.139,A 0.000,B 0.000,C 90.000,E1 24.951} C_DIS
LIN {X 0.007,Y -190.555,Z 822.116,A 0.000,B 0.000,C 90.000,E1 20.865} C_DIS
LIN {X 0.013,Y -186.787,Z 822.093,A 0.000,B 0.000,C 90.000,E1 16.732} C_DIS
LIN {X 0.070,Y -183.850,Z 822.065,A 0.000,B 0.000,C 90.000,E1 11.715} C_DIS
LIN {X 0.034,Y -184.694,Z 821.969,A 0.000,B 0.000,C 90.000,E1 354.489} C_DIS
LIN {X -0.054,Y -187.982,Z 821.942,A 0.000,B 0.000,C 90.000,E1 349.511} C_DIS
LIN {X 0.003,Y -191.662,Z 821.919,A 0.000,B 0.000,C 90.000,E1 345.353} C_DIS
LIN {X -0.092,Y -196.243,Z 821.896,A 0.000,B 0.000,C 90.000,E1 341.275} C_DIS
LIN {X 0.032,Y -201.708,Z 821.873,A 0.000,B 0.000,C 90.000,E1 337.177} C_DIS
LIN {X -0.012,Y -208.054,Z 821.851,A 0.000,B 0.000,C 90.000,E1 333.179} C_DIS
LIN {X 0.063,Y -215.292,Z 821.829,A 0.000,B 0.000,C 90.000,E1 329.203} C_DIS
LIN {X 0.050,Y -221.746,Z 821.812,A 0.000,B 0.000,C 90.000,E1 326.087} C_DIS
LIN {X -0.037,Y -230.524,Z 821.790,A 0.000,B 0.000,C 90.000,E1 322.271} C_DIS
LIN {X 0.070,Y -239.340,Z 821.771,A 0.000,B 0.000,C 90.000,E1 318.852} C_DIS
LIN {X -0.114,Y -248.848,Z 821.753,A 0.000,B 0.000,C 90.000,E1 315.567} C_DIS
LIN {X 0.131,Y -258.155,Z 821.737,A 0.000,B 0.000,C 90.000,E1 312.609} C_DIS
LIN {X -0.012,Y -269.262,Z 821.719,A 0.000,B 0.000,C 90.000,E1 309.439} C_DIS
LIN {X 0.026,Y -281.228,Z 821.702,A 0.000,B 0.000,C 90.000,E1 306.297} C_DIS
LIN {X 0.130,Y -295.963,Z 821.683,A 0.000,B 0.000,C 90.000,E1 302.880} C_DIS
LIN {X -0.087,Y -312.428,Z 821.664,A 0.000,B 0.000,C 90.000,E1 299.617} C_DIS
LIN {X 0.159,Y -327.144,Z 821.650,A 0.000,B 0.000,C 90.000,E1 297.001} C_DIS
LIN {X 0.044,Y -347.122,Z 821.633,A 0.000,B 0.000,C 90.000,E1 293.898} C_DIS
LIN {X 0.144,Y -364.889,Z 821.619,A 0.000,B 0.000,C 90.000,E1 291.461} C_DIS
LIN {X -0.130,Y -381.804,Z 821.608,A 0.000,B 0.000,C 90.000,E1 289.450} C_DIS
LIN {X 0.032,Y -399.530,Z 821.597,A 0.000,B 0.000,C 90.000,E1 287.457} C_DIS
LIN {X -0.107,Y -414.739,Z 821.588,A 0.000,B 0.000,C 90.000,E1 285.843} C_DIS
LIN {X 0.036,Y -427.166,Z 821.581,A 0.000,B 0.000,C 90.000,E1 284.481} C_DIS
LIN {X -0.044,Y -441.840,Z 821.572,A 0.000,B 0.000,C 90.000,E1 282.883} C_DIS
LIN {X 0.023,Y -450.993,Z 821.566,A 0.000,B 0.000,C 90.000,E1 281.827} C_DIS
LIN {X 0.065,Y -459.696,Z 821.560,A 0.000,B 0.000,C 90.000,E1 280.782} C_DIS
LIN {X -0.165,Y -467.628,Z 821.554,A 0.000,B 0.000,C 90.000,E1 279.782} C_DIS
LIN {X 0.216,Y -473.089,Z 821.550,A 0.000,B 0.000,C 90.000,E1 278.973} C_DIS
LIN {X 0.190,Y -478.046,Z 821.546,A 0.000,B 0.000,C 90.000,E1 278.219} C_DIS
LIN {X 0.136,Y -482.306,Z 821.542,A 0.000,B 0.000,C 90.000,E1 277.473} C_DIS
LIN {X 0.191,Y -485.929,Z 821.537,A 0.000,B 0.000,C 90.000,E1 276.720} C_DIS
LIN {X -0.218,Y -488.858,Z 821.533,A 0.000,B 0.000,C 90.000,E1 276.024} C_DIS
LIN {X -0.063,Y -490.359,Z 821.531,A 0.000,B 0.000,C 90.000,E1 275.511} C_DIS
LIN {X 0.155,Y -491.456,Z 821.528,A 0.000,B 0.000,C 90.000,E1 274.992} C_DIS
LIN {X -0.111,Y -492.241,Z 821.525,A 0.000,B 0.000,C 90.000,E1 274.531} C_DIS
LIN {X 0.119,Y -492.632,Z 821.522,A 0.000,B 0.000,C 90.000,E1 274.012} C_DIS
LIN {X -0.174,Y -492.630,Z 821.520,A 0.000,B 0.000,C 90.000,E1 273.555} C_DIS
LIN {X 0.059,Y -492.282,Z 821.517,A 0.000,B 0.000,C 90.000,E1 273.037} C_DIS
LIN {X -0.227,Y -491.495,Z 821.514,A 0.000,B 0.000,C 90.000,E1 272.579} C_DIS
LIN {X -0.021,Y -490.320,Z 821.511,A 0.000,B 0.000,C 90.000,E1 272.064} C_DIS
LIN {X 0.197,Y -488.749,Z 821.509,A 0.000,B 0.000,C 90.000,E1 271.547} C_DIS
LIN {X -0.096,Y -486.660,Z 821.506,A 0.000,B 0.000,C 90.000,E1 271.088} C_DIS
LIN {X 0.090,Y -484.028,Z 821.503,A 0.000,B 0.000,C 90.000,E1 270.573} C_DIS
LIN {X -0.224,Y -480.751,Z 821.500,A 0.000,B 0.000,C 90.000,E1 270.115} C_DIS
LIN {X -0.074,Y -476.764,Z 821.498,A 0.000,B 0.000,C 90.000,E1 269.599} C_DIS
LIN {X 0.053,Y -471.862,Z 821.495,A 0.000,B 0.000,C 90.000,E1 269.083} C_DIS
LIN {X -0.152,Y -466.147,Z 821.492,A 0.000,B 0.000,C 90.000,E1 268.625} C_DIS
LIN {X 0.084,Y -459.760,Z 821.490,A 0.000,B 0.000,C 90.000,E1 268.165} C_DIS
LIN {X -0.073,Y -452.741,Z 821.488,A 0.000,B 0.000,C 90.000,E1 267.822} C_DIS
LIN {X -0.095,Y -445.152,Z 821.486,A 0.000,B 0.000,C 90.000,E1 267.535} C_DIS
LIN {X -0.022,Y -437.180,Z 821.485,A 0.000,B 0.000,C 90.000,E1 267.306} C_DIS
LIN {X 0.076,Y -428.816,Z 821.484,A 0.000,B 0.000,C 90.000,E1 267.135} C_DIS
LIN {X -0.090,Y -419.496,Z 821.484,A 0.000,B 0.000,C 90.000,E1 267.078} C_DIS
LIN {X -0.066,Y -180.998,Z 821.484,A 0.000,B 0.000,C 90.000,E1 267.078} C_DIS
LIN {X -0.005,Y -180.863,Z 821.472,A 0.000,B 0.000,C 90.000,E1 265.008} C_DIS
LIN {X 0.049,Y -178.977,Z 821.444,A 0.000,B 0.000,C 90.000,E1 259.926} C_DIS
LIN {X 0.059,Y -177.943,Z 821.435,A 0.000,B 0.000,C 90.000,E1 258.229} C_DIS
LIN {X 0.073,Y -175.583,Z 821.411,A 0.000,B 0.000,C 90.000,E1 253.976} C_DIS
LIN {X 0.080,Y -172.309,Z 821.387,A 0.000,B 0.000,C 90.000,E1 249.699} C_DIS
LIN {X 0.057,Y -171.787,Z 821.383,A 0.000,B 0.000,C 90.000,E1 248.847} C_DIS
LIN {X -0.065,Y -169.455,Z 821.368,A 0.000,B 0.000,C 90.000,E1 246.305} C_DIS
LIN {X -0.009,Y -166.784,Z 821.349,A 0.000,B 0.000,C 90.000,E1 242.820} C_DIS
LIN {X -0.013,Y -162.764,Z 821.325,A 0.000,B 0.000,C 90.000,E1 238.456} C_DIS
LIN {X -0.038,Y -161.453,Z 821.315,A 0.000,B 0.000,C 90.000,E1 236.707} C_DIS
LIN {X 0.004,Y -157.447,Z 821.290,A 0.000,B 0.000,C 90.000,E1 232.271} C_DIS
LIN {X -0.063,Y -155.457,Z 821.276,A 0.000,B 0.000,C 90.000,E1 229.622} C_DIS
LIN {X -0.021,Y -151.773,Z 821.251,A 0.000,B 0.000,C 90.000,E1 225.121} C_DIS
LIN {X -0.004,Y -149.976,Z 821.236,A 0.000,B 0.000,C 90.000,E1 222.405} C_DIS
LIN {X 0.007,Y -146.812,Z 821.210,A 0.000,B 0.000,C 90.000,E1 217.855} C_DIS
LIN {X 0.023,Y -145.390,Z 821.195,A 0.000,B 0.000,C 90.000,E1 215.105} C_DIS
LIN {X -0.059,Y -142.827,Z 821.170,A 0.000,B 0.000,C 90.000,E1 210.541} C_DIS
LIN {X -0.002,Y -141.439,Z 821.149,A 0.000,B 0.000,C 90.000,E1 206.821} C_DIS
LIN {X 0.043,Y -139.368,Z 821.113,A 0.000,B 0.000,C 90.000,E1 200.301} C_DIS
LIN {X 0.028,Y -138.814,Z 821.097,A 0.000,B 0.000,C 90.000,E1 197.511} C_DIS
LIN {X -0.057,Y -138.351,Z 821.056,A 0.000,B 0.000,C 90.000,E1 190.074} C_DIS
LIN {X 0.056,Y -139.538,Z 821.004,A 0.000,B 0.000,C 90.000,E1 180.688} C_DIS
LIN {X 0.008,Y -141.229,Z 820.973,A 0.000,B 0.000,C 90.000,E1 175.122} C_DIS
LIN {X -0.033,Y -142.601,Z 820.957,A 0.000,B 0.000,C 90.000,E1 172.356} C_DIS
LIN {X 0.061,Y -144.907,Z 820.932,A 0.000,B 0.000,C 90.000,E1 167.701} C_DIS
LIN {X 0.014,Y -147.535,Z 820.911,A 0.000,B 0.000,C 90.000,E1 164.047} C_DIS
LIN {X -0.054,Y -150.135,Z 820.891,A 0.000,B 0.000,C 90.000,E1 160.423} C_DIS
LIN {X -0.043,Y -153.500,Z 820.871,A 0.000,B 0.000,C 90.000,E1 156.794} C_DIS
LIN {X 0.020,Y -157.865,Z 820.846,A 0.000,B 0.000,C 90.000,E1 152.281} C_DIS
LIN {X -0.025,Y -162.150,Z 820.826,A 0.000,B 0.000,C 90.000,E1 148.742} C_DIS
LIN {X 0.091,Y -166.356,Z 820.807,A 0.000,B 0.000,C 90.000,E1 145.182} C_DIS
LIN {X -0.040,Y -171.373,Z 820.787,A 0.000,B 0.000,C 90.000,E1 141.743} C_DIS
LIN {X 0.003,Y -176.282,Z 820.768,A 0.000,B 0.000,C 90.000,E1 138.286} C_DIS
LIN {X 0.003,Y -180.567,Z 820.754,A 0.000,B 0.000,C 90.000,E1 135.729} C_DIS
LIN {X -0.017,Y -185.968,Z 820.735,A 0.000,B 0.000,C 90.000,E1 132.366} C_DIS
LIN {X 0.038,Y -190.600,Z 820.721,A 0.000,B 0.000,C 90.000,E1 129.850} C_DIS
LIN {X 0.056,Y -192.776,Z 820.714,A 0.000,B 0.000,C 90.000,E1 128.543} C_DIS
LIN {X 0.056,Y -293.372,Z 820.714,A 0.000,B 0.000,C 90.000,E1 128.543} C_DIS
LIN {X -0.066,Y -294.758,Z 820.714,A 0.000,B 0.000,C 90.000,E1 128.543} C_DIS
LIN {X -0.066,Y -300.723,Z 820.712,A 0.000,B 0.000,C 90.000,E1 128.222} C_DIS
LIN {X -0.072,Y -303.812,Z 820.710,A 0.000,B 0.000,C 90.000,E1 127.890} C_DIS
LIN {X 0.046,Y -305.817,Z 820.709,A 0.000,B 0.000,C 90.000,E1 127.569} C_DIS
LIN {X -0.024,Y -307.387,Z 820.707,A 0.000,B 0.000,C 90.000,E1 127.282} C_DIS
LIN {X 0.002,Y -308.748,Z 820.705,A 0.000,B 0.000,C 90.000,E1 126.950} C_DIS
LIN {X 0.055,Y -313.643,Z 820.696,A 0.000,B 0.000,C 90.000,E1 125.311} C_DIS
LIN {X -0.138,Y -324.255,Z 820.678,A 0.000,B 0.000,C 90.000,E1 122.133} C_DIS
LIN {X -0.073,Y -335.164,Z 820.663,A 0.000,B 0.000,C 90.000,E1 119.283} C_DIS
LIN {X -0.015,Y -347.465,Z 820.647,A 0.000,B 0.000,C 90.000,E1 116.488} C_DIS
LIN {X -0.066,Y -361.261,Z 820.632,A 0.000,B 0.000,C 90.000,E1 113.770} C_DIS
LIN {X -0.119,Y -374.884,Z 820.619,A 0.000,B 0.000,C 90.000,E1 111.408} C_DIS
LIN {X -0.108,Y -389.887,Z 820.606,A 0.000,B 0.000,C 90.000,E1 109.087} C_DIS
LIN {X 0.032,Y -406.377,Z 820.593,A 0.000,B 0.000,C 90.000,E1 106.804} C_DIS
LIN {X 0.076,Y -424.474,Z 820.581,A 0.000,B 0.000,C 90.000,E1 104.592} C_DIS
LIN {X -0.023,Y -444.114,Z 820.569,A 0.000,B 0.000,C 90.000,E1 102.479} C_DIS
LIN {X 0.202,Y -464.460,Z 820.558,A 0.000,B 0.000,C 90.000,E1 100.489} C_DIS
LIN {X 0.211,Y -467.056,Z 820.557,A 0.000,B 0.000,C 90.000,E1 100.254} C_DIS
LIN {X 0.232,Y -469.268,Z 820.556,A 0.000,B 0.000,C 90.000,E1 100.018} C_DIS
LIN {X 0.172,Y -470.938,Z 820.555,A 0.000,B 0.000,C 90.000,E1 99.792} C_DIS
LIN {X 0.026,Y -472.318,Z 820.553,A 0.000,B 0.000,C 90.000,E1 99.557} C_DIS
LIN {X -0.122,Y -473.342,Z 820.552,A 0.000,B 0.000,C 90.000,E1 99.321} C_DIS
LIN {X -0.011,Y -474.521,Z 820.549,A 0.000,B 0.000,C 90.000,E1 98.803} C_DIS
LIN {X 0.179,Y -474.700,Z 820.546,A 0.000,B 0.000,C 90.000,E1 98.276} C_DIS
LIN {X -0.165,Y -473.911,Z 820.543,A 0.000,B 0.000,C 90.000,E1 97.814} C_DIS
LIN {X -0.036,Y -472.028,Z 820.541,A 0.000,B 0.000,C 90.000,E1 97.296} C_DIS
LIN {X 0.089,Y -468.883,Z 820.538,A 0.000,B 0.000,C 90.000,E1 96.777} C_DIS
LIN {X 0.164,Y -451.400,Z 820.522,A 0.000,B 0.000,C 90.000,E1 93.955} C_DIS
LIN {X -0.208,Y -440.831,Z 820.512,A 0.000,B 0.000,C 90.000,E1 92.178} C_DIS
LIN {X 0.215,Y -433.117,Z 820.505,A 0.000,B 0.000,C 90.000,E1 90.802} C_DIS
LIN {X -0.088,Y -421.859,Z 820.494,A 0.000,B 0.000,C 90.000,E1 88.969} C_DIS
LIN {X 0.139,Y -412.086,Z 820.485,A 0.000,B 0.000,C 90.000,E1 87.306} C_DIS
LIN {X -0.193,Y -402.167,Z 820.476,A 0.000,B 0.000,C 90.000,E1 85.698} C_DIS
LIN {X 0.207,Y -389.038,Z 820.463,A 0.000,B 0.000,C 90.000,E1 83.394} C_DIS
LIN {X -0.042,Y -374.568,Z 820.449,A 0.000,B 0.000,C 90.000,E1 80.849} C_DIS
LIN {X -0.175,Y -360.736,Z 820.434,A 0.000,B 0.000,C 90.000,E1 78.229} C_DIS
LIN {X -0.061,Y -350.409,Z 820.423,A 0.000,B 0.000,C 90.000,E1 76.117} C_DIS
LIN {X -0.097,Y -338.583,Z 820.409,A 0.000,B 0.000,C 90.000,E1 73.685} C_DIS
LIN {X 0.084,Y -326.947,Z 820.395,A 0.000,B 0.000,C 90.000,E1 71.167} C_DIS
LIN {X -0.005,Y -315.607,Z 820.381,A 0.000,B 0.000,C 90.000,E1 68.646} C_DIS
LIN {X -0.051,Y -303.365,Z 820.365,A 0.000,B 0.000,C 90.000,E1 65.741} C_DIS
LIN {X 0.053,Y -291.813,Z 820.349,A 0.000,B 0.000,C 90.000,E1 62.743} C_DIS
LIN {X -0.144,Y -280.658,Z 820.332,A 0.000,B 0.000,C 90.000,E1 59.744} C_DIS
LIN {X -0.080,Y -270.115,Z 820.315,A 0.000,B 0.000,C 90.000,E1 56.628} C_DIS
LIN {X 0.082,Y -261.221,Z 820.299,A 0.000,B 0.000,C 90.000,E1 53.783} C_DIS
LIN {X 0.041,Y -253.583,Z 820.285,A 0.000,B 0.000,C 90.000,E1 51.295} C_DIS
LIN {X 0.022,Y -245.186,Z 820.269,A 0.000,B 0.000,C 90.000,E1 48.405} C_DIS
LIN {X 0.024,Y -235.339,Z 820.248,A 0.000,B 0.000,C 90.000,E1 44.717} C_DIS
LIN {X -0.095,Y -226.347,Z 820.228,A 0.000,B 0.000,C 90.000,E1 40.987} C_DIS
LIN {X -0.091,Y -217.691,Z 820.206,A 0.000,B 0.000,C 90.000,E1 37.156} C_DIS
LIN {X 0.095,Y -211.083,Z 820.189,A 0.000,B 0.000,C 90.000,E1 33.992} C_DIS
LIN {X -0.056,Y -205.064,Z 820.171,A 0.000,B 0.000,C 90.000,E1 30.875} C_DIS
LIN {X 0.067,Y -199.661,Z 820.154,A 0.000,B 0.000,C 90.000,E1 27.641} C_DIS
LIN {X 0.125,Y -195.032,Z 820.136,A 0.000,B 0.000,C 90.000,E1 24.387} C_DIS
LIN {X 0.104,Y -190.306,Z 820.113,A 0.000,B 0.000,C 90.000,E1 20.301} C_DIS
LIN {X -0.017,Y -186.692,Z 820.090,A 0.000,B 0.000,C 90.000,E1 16.205} C_DIS
LIN {X 0.043,Y -183.911,Z 820.062,A 0.000,B 0.000,C 90.000,E1 11.186} C_DIS
LIN {X 0.044,Y -184.948,Z 819.969,A 0.000,B 0.000,C 90.000,E1 354.489} C_DIS
LIN {X -0.035,Y -188.219,Z 819.942,A 0.000,B 0.000,C 90.000,E1 349.511} C_DIS
LIN {X 0.030,Y -191.862,Z 819.919,A 0.000,B 0.000,C 90.000,E1 345.353} C_DIS
LIN {X -0.057,Y -196.439,Z 819.896,A 0.000,B 0.000,C 90.000,E1 341.275} C_DIS
LIN {X 0.074,Y -201.894,Z 819.873,A 0.000,B 0.000,C 90.000,E1 337.177} C_DIS
LIN {X 0.036,Y -208.236,Z 819.851,A 0.000,B 0.000,C 90.000,E1 333.179} C_DIS
LIN {X 0.081,Y -213.949,Z 819.833,A 0.000,B 0.000,C 90.000,E1 329.999} C_DIS
LIN {X -0.081,Y -220.268,Z 819.816,A 0.000,B 0.000,C 90.000,E1 326.914} C_DIS
LIN {X -0.034,Y -228.917,Z 819.795,A 0.000,B 0.000,C 90.000,E1 323.050} C_DIS
LIN {X 0.089,Y -236.478,Z 819.778,A 0.000,B 0.000,C 90.000,E1 319.989} C_DIS
LIN {X -0.007,Y -246.819,Z 819.757,A 0.000,B 0.000,C 90.000,E1 316.296} C_DIS
LIN {X 0.025,Y -257.098,Z 819.739,A 0.000,B 0.000,C 90.000,E1 313.014} C_DIS
LIN {X 0.020,Y -268.039,Z 819.721,A 0.000,B 0.000,C 90.000,E1 309.806} C_DIS
LIN {X 0.029,Y -279.845,Z 819.704,A 0.000,B 0.000,C 90.000,E1 306.664} C_DIS
LIN {X 0.094,Y -294.387,Z 819.685,A 0.000,B 0.000,C 90.000,E1 303.245} C_DIS
LIN {X -0.010,Y -310.631,Z 819.666,A 0.000,B 0.000,C 90.000,E1 299.951} C_DIS
LIN {X -0.095,Y -325.104,Z 819.652,A 0.000,B 0.000,C 90.000,E1 297.385} C_DIS
LIN {X 0.034,Y -340.760,Z 819.638,A 0.000,B 0.000,C 90.000,E1 294.847} C_DIS
LIN {X -0.066,Y -355.579,Z 819.626,A 0.000,B 0.000,C 90.000,E1 292.717} C_DIS
LIN {X 0.112,Y -374.128,Z 819.613,A 0.000,B 0.000,C 90.000,E1 290.301} C_DIS
LIN {X -0.037,Y -391.682,Z 819.602,A 0.000,B 0.000,C 90.000,E1 288.308} C_DIS
LIN {X -0.095,Y -409.592,Z 819.591,A 0.000,B 0.000,C 90.000,E1 286.370} C_DIS
LIN {X 0.037,Y -422.099,Z 819.583,A 0.000,B 0.000,C 90.000,E1 285.009} C_DIS
LIN {X -0.062,Y -434.146,Z 819.576,A 0.000,B 0.000,C 90.000,E1 283.703} C_DIS
LIN {X -0.137,Y -443.844,Z 819.570,A 0.000,B 0.000,C 90.000,E1 282.647} C_DIS
LIN {X -0.097,Y -452.919,Z 819.564,A 0.000,B 0.000,C 90.000,E1 281.591} C_DIS
LIN {X -0.036,Y -461.449,Z 819.559,A 0.000,B 0.000,C 90.000,E1 280.546} C_DIS
LIN {X 0.134,Y -469.249,Z 819.553,A 0.000,B 0.000,C 90.000,E1 279.500} C_DIS
LIN {X 0.077,Y -474.571,Z 819.549,A 0.000,B 0.000,C 90.000,E1 278.746} C_DIS
LIN {X 0.060,Y -479.279,Z 819.544,A 0.000,B 0.000,C 90.000,E1 277.992} C_DIS
LIN {X 0.087,Y -483.393,Z 819.540,A 0.000,B 0.000,C 90.000,E1 277.239} C_DIS
LIN {X 0.143,Y -486.841,Z 819.536,A 0.000,B 0.000,C 90.000,E1 276.486} C_DIS
LIN {X -0.145,Y -488.728,Z 819.533,A 0.000,B 0.000,C 90.000,E1 276.024} C_DIS
LIN {X 0.009,Y -490.282,Z 819.531,A 0.000,B 0.000,C 90.000,E1 275.511} C_DIS
LIN {X 0.226,Y -491.426,Z 819.528,A 0.000,B 0.000,C 90.000,E1 274.992} C_DIS
LIN {X -0.040,Y -492.212,Z 819.525,A 0.000,B 0.000,C 90.000,E1 274.531} C_DIS
LIN {X 0.189,Y -492.618,Z 819.522,A 0.000,B 0.000,C 90.000,E1 274.012} C_DIS
LIN {X -0.104,Y -492.633,Z 819.520,A 0.000,B 0.000,C 90.000,E1 273.555} C_DIS
LIN {X 0.128,Y -492.290,Z 819.517,A 0.000,B 0.000,C 90.000,E1 273.037} C_DIS
LIN {X -0.157,Y -491.532,Z 819.514,A 0.000,B 0.000,C 90.000,E1 272.579} C_DIS
LIN {X 0.049,Y -490.375,Z 819.511,A 0.000,B 0.000,C 90.000,E1 272.064} C_DIS
LIN {X -0.222,Y -488.819,Z 819.509,A 0.000,B 0.000,C 90.000,E1 271.604} C_DIS
LIN {X -0.026,Y -486.768,Z 819.506,A 0.000,B 0.000,C 90.000,E1 271.088} C_DIS
LIN {X 0.160,Y -484.196,Z 819.503,A 0.000,B 0.000,C 90.000,E1 270.573} C_DIS
LIN {X -0.155,Y -480.968,Z 819.501,A 0.000,B 0.000,C 90.000,E1 270.115} C_DIS
LIN {X -0.004,Y -477.045,Z 819.498,A 0.000,B 0.000,C 90.000,E1 269.599} C_DIS
LIN {X 0.125,Y -472.189,Z 819.495,A 0.000,B 0.000,C 90.000,E1 269.083} C_DIS
LIN {X -0.116,Y -466.515,Z 819.492,A 0.000,B 0.000,C 90.000,E1 268.625} C_DIS
LIN {X 0.092,Y -460.205,Z 819.490,A 0.000,B 0.000,C 90.000,E1 268.165} C_DIS
LIN {X -0.015,Y -456.958,Z 819.489,A 0.000,B 0.000,C 90.000,E1 267.993} C_DIS
LIN {X 0.103,Y -449.662,Z 819.487,A 0.000,B 0.000,C 90.000,E1 267.650} C_DIS
LIN {X -0.090,Y -442.114,Z 819.486,A 0.000,B 0.000,C 90.000,E1 267.421} C_DIS
LIN {X 0.196,Y -434.309,Z 819.485,A 0.000,B 0.000,C 90.000,E1 267.192} C_DIS
LIN {X 0.105,Y -425.836,Z 819.484,A 0.000,B 0.000,C 90.000,E1 267.078} C_DIS
LIN {X 0.146,Y -417.403,Z 819.484,A 0.000,B 0.000,C 90.000,E1 267.020} C_DIS
LIN {X 0.036,Y -180.995,Z 819.484,A 0.000,B 0.000,C 90.000,E1 267.020} C_DIS
LIN {X -0.028,Y -180.861,Z 819.472,A 0.000,B 0.000,C 90.000,E1 265.008} C_DIS
LIN {X 0.026,Y -178.975,Z 819.444,A 0.000,B 0.000,C 90.000,E1 259.926} C_DIS
LIN {X 0.036,Y -177.937,Z 819.435,A 0.000,B 0.000,C 90.000,E1 258.229} C_DIS
LIN {X 0.051,Y -175.577,Z 819.411,A 0.000,B 0.000,C 90.000,E1 253.976} C_DIS
LIN {X 0.057,Y -172.303,Z 819.387,A 0.000,B 0.000,C 90.000,E1 249.699} C_DIS
LIN {X 0.035,Y -171.783,Z 819.383,A 0.000,B 0.000,C 90.000,E1 248.847} C_DIS
LIN {X -0.020,Y -169.448,Z 819.368,A 0.000,B 0.000,C 90.000,E1 246.282} C_DIS
LIN {X 0.045,Y -166.778,Z 819.349,A 0.000,B 0.000,C 90.000,E1 242.794} C_DIS
LIN {X -0.035,Y -162.758,Z 819.325,A 0.000,B 0.000,C 90.000,E1 238.456} C_DIS
LIN {X -0.059,Y -161.448,Z 819.315,A 0.000,B 0.000,C 90.000,E1 236.707} C_DIS
LIN {X -0.018,Y -157.441,Z 819.290,A 0.000,B 0.000,C 90.000,E1 232.271} C_DIS
LIN {X 0.017,Y -155.449,Z 819.276,A 0.000,B 0.000,C 90.000,E1 229.585} C_DIS
LIN {X 0.065,Y -151.767,Z 819.251,A 0.000,B 0.000,C 90.000,E1 225.081} C_DIS
LIN {X 0.076,Y -149.970,Z 819.236,A 0.000,B 0.000,C 90.000,E1 222.366} C_DIS
LIN {X -0.014,Y -146.808,Z 819.210,A 0.000,B 0.000,C 90.000,E1 217.855} C_DIS
LIN {X 0.003,Y -145.385,Z 819.195,A 0.000,B 0.000,C 90.000,E1 215.105} C_DIS
LIN {X -0.006,Y -142.443,Z 819.164,A 0.000,B 0.000,C 90.000,E1 209.589} C_DIS
LIN {X -0.022,Y -141.435,Z 819.149,A 0.000,B 0.000,C 90.000,E1 206.821} C_DIS
LIN {X 0.023,Y -139.366,Z 819.113,A 0.000,B 0.000,C 90.000,E1 200.301} C_DIS
LIN {X 0.009,Y -138.812,Z 819.097,A 0.000,B 0.000,C 90.000,E1 197.511} C_DIS
LIN {X 0.060,Y -138.352,Z 819.056,A 0.000,B 0.000,C 90.000,E1 190.018} C_DIS
LIN {X 0.036,Y -139.539,Z 819.004,A 0.000,B 0.000,C 90.000,E1 180.688} C_DIS
LIN {X -0.012,Y -141.233,Z 818.973,A 0.000,B 0.000,C 90.000,E1 175.122} C_DIS
LIN {X -0.053,Y -142.603,Z 818.957,A 0.000,B 0.000,C 90.000,E1 172.356} C_DIS
LIN {X 0.042,Y -144.912,Z 818.932,A 0.000,B 0.000,C 90.000,E1 167.701} C_DIS
LIN {X 0.034,Y -147.540,Z 818.911,A 0.000,B 0.000,C 90.000,E1 164.031} C_DIS
LIN {X 0.067,Y -150.141,Z 818.891,A 0.000,B 0.000,C 90.000,E1 160.369} C_DIS
LIN {X -0.064,Y -153.508,Z 818.871,A 0.000,B 0.000,C 90.000,E1 156.794} C_DIS
LIN {X -0.002,Y -157.873,Z 818.846,A 0.000,B 0.000,C 90.000,E1 152.281} C_DIS
LIN {X -0.047,Y -162.160,Z 818.826,A 0.000,B 0.000,C 90.000,E1 148.742} C_DIS
LIN {X 0.068,Y -166.366,Z 818.807,A 0.000,B 0.000,C 90.000,E1 145.182} C_DIS
LIN {X -0.063,Y -171.383,Z 818.787,A 0.000,B 0.000,C 90.000,E1 141.743} C_DIS
LIN {X 0.111,Y -176.293,Z 818.768,A 0.000,B 0.000,C 90.000,E1 138.243} C_DIS
LIN {X -0.020,Y -180.579,Z 818.754,A 0.000,B 0.000,C 90.000,E1 135.729} C_DIS
LIN {X -0.041,Y -185.981,Z 818.735,A 0.000,B 0.000,C 90.000,E1 132.366} C_DIS
LIN {X 0.015,Y -190.614,Z 818.721,A 0.000,B 0.000,C 90.000,E1 129.850} C_DIS
LIN {X 0.092,Y -192.758,Z 818.714,A 0.000,B 0.000,C 90.000,E1 128.543} C_DIS
LIN {X 0.111,Y -293.048,Z 818.714,A 0.000,B 0.000,C 90.000,E1 128.543} C_DIS
LIN {X -0.101,Y -295.288,Z 818.714,A 0.000,B 0.000,C 90.000,E1 128.543} C_DIS
LIN {X 0.133,Y -300.855,Z 818.712,A 0.000,B 0.000,C 90.000,E1 128.177} C_DIS
LIN {X -0.040,Y -304.050,Z 818.710,A 0.000,B 0.000,C 90.000,E1 127.855} C_DIS
LIN {X 0.095,Y -306.029,Z 818.709,A 0.000,B 0.000,C 90.000,E1 127.523} C_DIS
LIN {X -0.011,Y -307.579,Z 818.707,A 0.000,B 0.000,C 90.000,E1 127.237} C_DIS
LIN {X -0.045,Y -308.889,Z 818.705,A 0.000,B 0.000,C 90.000,E1 126.916} C_DIS
LIN {X -0.080,Y -321.033,Z 818.683,A 0.000,B 0.000,C 90.000,E1 123.038} C_DIS
LIN {X -0.054,Y -331.521,Z 818.668,A 0.000,B 0.000,C 90.000,E1 120.178} C_DIS
LIN {X -0.107,Y -343.364,Z 818.652,A 0.000,B 0.000,C 90.000,E1 117.385} C_DIS
LIN {X -0.134,Y -356.674,Z 818.637,A 0.000,B 0.000,C 90.000,E1 114.643} C_DIS
LIN {X 0.176,Y -369.827,Z 818.624,A 0.000,B 0.000,C 90.000,E1 112.206} C_DIS
LIN {X 0.069,Y -384.324,Z 818.611,A 0.000,B 0.000,C 90.000,E1 109.885} C_DIS
LIN {X -0.179,Y -400.268,Z 818.598,A 0.000,B 0.000,C 90.000,E1 107.638} C_DIS
LIN {X 0.106,Y -417.774,Z 818.585,A 0.000,B 0.000,C 90.000,E1 105.371} C_DIS
LIN {X -0.183,Y -436.949,Z 818.573,A 0.000,B 0.000,C 90.000,E1 103.244} C_DIS
LIN {X 0.080,Y -457.095,Z 818.562,A 0.000,B 0.000,C 90.000,E1 101.186} C_DIS
LIN {X -0.044,Y -467.365,Z 818.557,A 0.000,B 0.000,C 90.000,E1 100.254} C_DIS
LIN {X -0.026,Y -469.500,Z 818.556,A 0.000,B 0.000,C 90.000,E1 100.018} C_DIS
LIN {X -0.088,Y -471.117,Z 818.554,A 0.000,B 0.000,C 90.000,E1 99.792} C_DIS
LIN {X -0.235,Y -472.452,Z 818.553,A 0.000,B 0.000,C 90.000,E1 99.557} C_DIS
LIN {X 0.084,Y -473.439,Z 818.552,A 0.000,B 0.000,C 90.000,E1 99.265} C_DIS
LIN {X 0.197,Y -474.557,Z 818.549,A 0.000,B 0.000,C 90.000,E1 98.746} C_DIS
LIN {X -0.081,Y -474.681,Z 818.546,A 0.000,B 0.000,C 90.000,E1 98.276} C_DIS
LIN {X 0.045,Y -473.835,Z 818.543,A 0.000,B 0.000,C 90.000,E1 97.757} C_DIS
LIN {X 0.174,Y -471.881,Z 818.540,A 0.000,B 0.000,C 90.000,E1 97.239} C_DIS
LIN {X 0.142,Y -467.028,Z 818.536,A 0.000,B 0.000,C 90.000,E1 96.486} C_DIS
LIN {X -0.121,Y -448.243,Z 818.519,A 0.000,B 0.000,C 90.000,E1 93.440} C_DIS
LIN {X -0.089,Y -437.619,Z 818.509,A 0.000,B 0.000,C 90.000,E1 91.604} C_DIS
LIN {X -0.159,Y -429.762,Z 818.501,A 0.000,B 0.000,C 90.000,E1 90.286} C_DIS
LIN {X -0.100,Y -418.481,Z 818.491,A 0.000,B 0.000,C 90.000,E1 88.396} C_DIS
LIN {X 0.084,Y -408.643,Z 818.482,A 0.000,B 0.000,C 90.000,E1 86.731} C_DIS
LIN {X 0.134,Y -397.078,Z 818.471,A 0.000,B 0.000,C 90.000,E1 84.780} C_DIS
LIN {X 0.008,Y -384.033,Z 818.459,A 0.000,B 0.000,C 90.000,E1 82.534} C_DIS
LIN {X 0.052,Y -369.773,Z 818.444,A 0.000,B 0.000,C 90.000,E1 79.926} C_DIS
LIN {X 0.174,Y -353.232,Z 818.426,A 0.000,B 0.000,C 90.000,E1 76.645} C_DIS
LIN {X -0.129,Y -342.891,Z 818.414,A 0.000,B 0.000,C 90.000,E1 74.574} C_DIS
LIN {X -0.130,Y -332.663,Z 818.402,A 0.000,B 0.000,C 90.000,E1 72.417} C_DIS
LIN {X 0.015,Y -321.188,Z 818.388,A 0.000,B 0.000,C 90.000,E1 69.880} C_DIS
LIN {X 0.083,Y -310.066,Z 818.374,A 0.000,B 0.000,C 90.000,E1 67.305} C_DIS
LIN {X 0.120,Y -296.888,Z 818.356,A 0.000,B 0.000,C 90.000,E1 64.024} C_DIS
LIN {X -0.058,Y -286.857,Z 818.341,A 0.000,B 0.000,C 90.000,E1 61.385} C_DIS
LIN {X -0.160,Y -274.893,Z 818.322,A 0.000,B 0.000,C 90.000,E1 57.995} C_DIS
LIN {X -0.043,Y -263.613,Z 818.303,A 0.000,B 0.000,C 90.000,E1 54.482} C_DIS
LIN {X 0.023,Y -255.982,Z 818.289,A 0.000,B 0.000,C 90.000,E1 51.984} C_DIS
LIN {X -0.106,Y -245.432,Z 818.269,A 0.000,B 0.000,C 90.000,E1 48.405} C_DIS
LIN {X 0.078,Y -235.594,Z 818.248,A 0.000,B 0.000,C 90.000,E1 44.676} C_DIS
LIN {X -0.026,Y -226.610,Z 818.227,A 0.000,B 0.000,C 90.000,E1 40.943} C_DIS
LIN {X -0.039,Y -219.650,Z 818.210,A 0.000,B 0.000,C 90.000,E1 37.890} C_DIS
LIN {X 0.014,Y -211.359,Z 818.189,A 0.000,B 0.000,C 90.000,E1 33.992} C_DIS
LIN {X -0.023,Y -205.344,Z 818.171,A 0.000,B 0.000,C 90.000,E1 30.846} C_DIS
LIN {X 0.005,Y -199.956,Z 818.154,A 0.000,B 0.000,C 90.000,E1 27.641} C_DIS
LIN {X 0.071,Y -195.303,Z 818.136,A 0.000,B 0.000,C 90.000,E1 24.387} C_DIS
LIN {X 0.060,Y -190.579,Z 818.113,A 0.000,B 0.000,C 90.000,E1 20.301} C_DIS
LIN {X -0.052,Y -186.973,Z 818.090,A 0.000,B 0.000,C 90.000,E1 16.205} C_DIS
LIN {X 0.018,Y -184.196,Z 818.062,A 0.000,B 0.000,C 90.000,E1 11.186} C_DIS
LIN {X 0.055,Y -185.204,Z 817.969,A 0.000,B 0.000,C 90.000,E1 354.489} C_DIS
LIN {X -0.014,Y -188.449,Z 817.942,A 0.000,B 0.000,C 90.000,E1 349.511} C_DIS
LIN {X 0.057,Y -192.056,Z 817.919,A 0.000,B 0.000,C 90.000,E1 345.353} C_DIS
LIN {X -0.023,Y -196.633,Z 817.896,A 0.000,B 0.000,C 90.000,E1 341.275} C_DIS
LIN {X -0.071,Y -202.079,Z 817.873,A 0.000,B 0.000,C 90.000,E1 337.230} C_DIS
LIN {X -0.010,Y -208.391,Z 817.851,A 0.000,B 0.000,C 90.000,E1 333.204} C_DIS
LIN {X -0.051,Y -214.135,Z 817.834,A 0.000,B 0.000,C 90.000,E1 330.049} C_DIS
LIN {X -0.009,Y -222.129,Z 817.812,A 0.000,B 0.000,C 90.000,E1 326.135} C_DIS
LIN {X 0.034,Y -229.109,Z 817.795,A 0.000,B 0.000,C 90.000,E1 323.050} C_DIS
LIN {X -0.051,Y -237.652,Z 817.776,A 0.000,B 0.000,C 90.000,E1 319.666} C_DIS
LIN {X 0.078,Y -246.973,Z 817.757,A 0.000,B 0.000,C 90.000,E1 316.296} C_DIS
LIN {X -0.071,Y -257.210,Z 817.739,A 0.000,B 0.000,C 90.000,E1 313.056} C_DIS
LIN {X -0.087,Y -268.100,Z 817.721,A 0.000,B 0.000,C 90.000,E1 309.850} C_DIS
LIN {X 0.134,Y -279.858,Z 817.704,A 0.000,B 0.000,C 90.000,E1 306.664} C_DIS
LIN {X -0.043,Y -294.354,Z 817.685,A 0.000,B 0.000,C 90.000,E1 303.293} C_DIS
LIN {X -0.164,Y -310.563,Z 817.667,A 0.000,B 0.000,C 90.000,E1 300.001} C_DIS
LIN {X -0.040,Y -326.907,Z 817.650,A 0.000,B 0.000,C 90.000,E1 297.078} C_DIS
LIN {X -0.026,Y -346.767,Z 817.633,A 0.000,B 0.000,C 90.000,E1 293.951} C_DIS
LIN {X -0.135,Y -362.114,Z 817.621,A 0.000,B 0.000,C 90.000,E1 291.844} C_DIS
LIN {X 0.037,Y -378.681,Z 817.610,A 0.000,B 0.000,C 90.000,E1 289.758} C_DIS
LIN {X -0.154,Y -393.926,Z 817.600,A 0.000,B 0.000,C 90.000,E1 288.055} C_DIS
LIN {X -0.056,Y -409.190,Z 817.591,A 0.000,B 0.000,C 90.000,E1 286.386} C_DIS
LIN {X 0.200,Y -421.682,Z 817.584,A 0.000,B 0.000,C 90.000,E1 285.009} C_DIS
LIN {X -0.110,Y -433.976,Z 817.576,A 0.000,B 0.000,C 90.000,E1 283.703} C_DIS
LIN {X -0.162,Y -443.642,Z 817.570,A 0.000,B 0.000,C 90.000,E1 282.647} C_DIS
LIN {X -0.126,Y -452.719,Z 817.564,A 0.000,B 0.000,C 90.000,E1 281.591} C_DIS
LIN {X -0.067,Y -461.256,Z 817.559,A 0.000,B 0.000,C 90.000,E1 280.546} C_DIS
LIN {X 0.100,Y -469.051,Z 817.553,A 0.000,B 0.000,C 90.000,E1 279.500} C_DIS
LIN {X 0.041,Y -474.407,Z 817.549,A 0.000,B 0.000,C 90.000,E1 278.746} C_DIS
LIN {X 0.022,Y -479.137,Z 817.544,A 0.000,B 0.000,C 90.000,E1 277.992} C_DIS
LIN {X 0.047,Y -483.253,Z 817.540,A 0.000,B 0.000,C 90.000,E1 277.239} C_DIS
LIN {X 0.101,Y -486.742,Z 817.536,A 0.000,B 0.000,C 90.000,E1 276.486} C_DIS
LIN {X -0.188,Y -488.639,Z 817.533,A 0.000,B 0.000,C 90.000,E1 276.024} C_DIS
LIN {X -0.034,Y -490.229,Z 817.531,A 0.000,B 0.000,C 90.000,E1 275.511} C_DIS
LIN {X 0.183,Y -491.417,Z 817.528,A 0.000,B 0.000,C 90.000,E1 274.992} C_DIS
LIN {X -0.083,Y -492.174,Z 817.525,A 0.000,B 0.000,C 90.000,E1 274.531} C_DIS
LIN {X 0.145,Y -492.602,Z 817.522,A 0.000,B 0.000,C 90.000,E1 274.012} C_DIS
LIN {X -0.148,Y -492.644,Z 817.520,A 0.000,B 0.000,C 90.000,E1 273.555} C_DIS
LIN {X 0.084,Y -492.290,Z 817.517,A 0.000,B 0.000,C 90.000,E1 273.037} C_DIS
LIN {X -0.201,Y -491.558,Z 817.514,A 0.000,B 0.000,C 90.000,E1 272.579} C_DIS
LIN {X 0.005,Y -490.402,Z 817.511,A 0.000,B 0.000,C 90.000,E1 272.064} C_DIS
LIN {X 0.223,Y -488.839,Z 817.509,A 0.000,B 0.000,C 90.000,E1 271.547} C_DIS
LIN {X -0.070,Y -486.832,Z 817.506,A 0.000,B 0.000,C 90.000,E1 271.088} C_DIS
LIN {X 0.116,Y -484.275,Z 817.503,A 0.000,B 0.000,C 90.000,E1 270.573} C_DIS
LIN {X -0.197,Y -481.069,Z 817.500,A 0.000,B 0.000,C 90.000,E1 270.115} C_DIS
LIN {X -0.045,Y -477.189,Z 817.498,A 0.000,B 0.000,C 90.000,E1 269.599} C_DIS
LIN {X 0.084,Y -472.387,Z 817.495,A 0.000,B 0.000,C 90.000,E1 269.083} C_DIS
LIN {X -0.047,Y -469.729,Z 817.494,A 0.000,B 0.000,C 90.000,E1 268.854} C_DIS
LIN {X -0.072,Y -463.780,Z 817.491,A 0.000,B 0.000,C 90.000,E1 268.396} C_DIS
LIN {X -0.063,Y -457.267,Z 817.489,A 0.000,B 0.000,C 90.000,E1 267.993} C_DIS
LIN {X -0.170,Y -453.489,Z 817.488,A 0.000,B 0.000,C 90.000,E1 267.822} C_DIS
LIN {X -0.216,Y -445.974,Z 817.486,A 0.000,B 0.000,C 90.000,E1 267.535} C_DIS
LIN {X -0.171,Y -438.007,Z 817.485,A 0.000,B 0.000,C 90.000,E1 267.306} C_DIS
LIN {X -0.093,Y -430.047,Z 817.484,A 0.000,B 0.000,C 90.000,E1 267.135} C_DIS
LIN {X 0.163,Y -422.755,Z 817.484,A 0.000,B 0.000,C 90.000,E1 267.020} C_DIS
LIN {X 0.035,Y -418.079,Z 817.483,A 0.000,B 0.000,C 90.000,E1 267.020} C_DIS
LIN {X -0.013,Y -180.993,Z 817.483,A 0.000,B 0.000,C 90.000,E1 267.020} C_DIS
LIN {X -0.078,Y -180.858,Z 817.472,A 0.000,B 0.000,C 90.000,E1 265.008} C_DIS
LIN {X -0.024,Y -178.970,Z 817.444,A 0.000,B 0.000,C 90.000,E1 259.926} C_DIS
LIN {X -0.013,Y -177.927,Z 817.435,A 0.000,B 0.000,C 90.000,E1 258.229} C_DIS
LIN {X 0.001,Y -175.565,Z 817.411,A 0.000,B 0.000,C 90.000,E1 253.976} C_DIS
LIN {X 0.008,Y -172.294,Z 817.387,A 0.000,B 0.000,C 90.000,E1 249.699} C_DIS
LIN {X -0.014,Y -171.773,Z 817.382,A 0.000,B 0.000,C 90.000,E1 248.847} C_DIS
LIN {X -0.041,Y -168.700,Z 817.363,A 0.000,B 0.000,C 90.000,E1 245.409} C_DIS
LIN {X -0.003,Y -166.765,Z 817.349,A 0.000,B 0.000,C 90.000,E1 242.794} C_DIS
LIN {X 0.056,Y -162.745,Z 817.325,A 0.000,B 0.000,C 90.000,E1 238.408} C_DIS
LIN {X -0.106,Y -161.434,Z 817.315,A 0.000,B 0.000,C 90.000,E1 236.707} C_DIS
LIN {X -0.063,Y -157.428,Z 817.290,A 0.000,B 0.000,C 90.000,E1 232.271} C_DIS
LIN {X -0.029,Y -155.434,Z 817.275,A 0.000,B 0.000,C 90.000,E1 229.585} C_DIS
LIN {X 0.020,Y -151.755,Z 817.250,A 0.000,B 0.000,C 90.000,E1 225.081} C_DIS
LIN {X 0.032,Y -149.956,Z 817.235,A 0.000,B 0.000,C 90.000,E1 222.366} C_DIS
LIN {X 0.059,Y -146.798,Z 817.210,A 0.000,B 0.000,C 90.000,E1 217.810} C_DIS
LIN {X -0.041,Y -145.374,Z 817.195,A 0.000,B 0.000,C 90.000,E1 215.105} C_DIS
LIN {X 0.076,Y -142.437,Z 817.164,A 0.000,B 0.000,C 90.000,E1 209.539} C_DIS
LIN {X -0.001,Y -141.427,Z 817.149,A 0.000,B 0.000,C 90.000,E1 206.796} C_DIS
LIN {X -0.020,Y -139.364,Z 817.113,A 0.000,B 0.000,C 90.000,E1 200.301} C_DIS
LIN {X -0.034,Y -138.808,Z 817.097,A 0.000,B 0.000,C 90.000,E1 197.511} C_DIS
LIN {X 0.017,Y -138.350,Z 817.056,A 0.000,B 0.000,C 90.000,E1 190.018} C_DIS
LIN {X -0.007,Y -139.542,Z 817.004,A 0.000,B 0.000,C 90.000,E1 180.688} C_DIS
LIN {X -0.055,Y -141.240,Z 816.973,A 0.000,B 0.000,C 90.000,E1 175.122} C_DIS
LIN {X 0.045,Y -142.610,Z 816.957,A 0.000,B 0.000,C 90.000,E1 172.299} C_DIS
LIN {X -0.003,Y -144.923,Z 816.932,A 0.000,B 0.000,C 90.000,E1 167.701} C_DIS
LIN {X -0.010,Y -147.552,Z 816.911,A 0.000,B 0.000,C 90.000,E1 164.031} C_DIS
LIN {X 0.022,Y -150.155,Z 816.891,A 0.000,B 0.000,C 90.000,E1 160.369} C_DIS
LIN {X 0.031,Y -153.526,Z 816.871,A 0.000,B 0.000,C 90.000,E1 156.741} C_DIS
LIN {X 0.084,Y -156.944,Z 816.851,A 0.000,B 0.000,C 90.000,E1 153.127} C_DIS
LIN {X 0.020,Y -161.047,Z 816.831,A 0.000,B 0.000,C 90.000,E1 149.587} C_DIS
LIN {X 0.105,Y -163.157,Z 816.821,A 0.000,B 0.000,C 90.000,E1 147.788} C_DIS
LIN {X -0.024,Y -167.573,Z 816.802,A 0.000,B 0.000,C 90.000,E1 144.322} C_DIS
LIN {X 0.022,Y -171.404,Z 816.787,A 0.000,B 0.000,C 90.000,E1 141.698} C_DIS
LIN {X 0.062,Y -176.319,Z 816.768,A 0.000,B 0.000,C 90.000,E1 138.243} C_DIS
LIN {X -0.070,Y -180.607,Z 816.754,A 0.000,B 0.000,C 90.000,E1 135.729} C_DIS
LIN {X 0.045,Y -186.009,Z 816.735,A 0.000,B 0.000,C 90.000,E1 132.324} C_DIS
LIN {X -0.038,Y -190.643,Z 816.721,A 0.000,B 0.000,C 90.000,E1 129.850} C_DIS
LIN {X -0.018,Y -192.737,Z 816.714,A 0.000,B 0.000,C 90.000,E1 128.588} C_DIS
LIN {X -0.062,Y -292.570,Z 816.714,A 0.000,B 0.000,C 90.000,E1 128.588} C_DIS
LIN {X 0.064,Y -294.292,Z 816.714,A 0.000,B 0.000,C 90.000,E1 128.543} C_DIS
LIN {X -0.059,Y -298.710,Z 816.713,A 0.000,B 0.000,C 90.000,E1 128.382} C_DIS
LIN {X 0.051,Y -301.076,Z 816.712,A 0.000,B 0.000,C 90.000,E1 128.177} C_DIS
LIN {X -0.030,Y -304.924,Z 816.710,A 0.000,B 0.000,C 90.000,E1 127.729} C_DIS
LIN {X 0.009,Y -306.790,Z 816.708,A 0.000,B 0.000,C 90.000,E1 127.397} C_DIS
LIN {X -0.008,Y -308.249,Z 816.706,A 0.000,B 0.000,C 90.000,E1 127.076} C_DIS
LIN {X -0.013,Y -310.354,Z 816.702,A 0.000,B 0.000,C 90.000,E1 126.423} C_DIS
LIN {X 0.122,Y -320.455,Z 816.684,A 0.000,B 0.000,C 90.000,E1 123.166} C_DIS
LIN {X -0.028,Y -330.867,Z 816.669,A 0.000,B 0.000,C 90.000,E1 120.335} C_DIS
LIN {X 0.067,Y -342.634,Z 816.653,A 0.000,B 0.000,C 90.000,E1 117.513} C_DIS
LIN {X 0.030,Y -355.854,Z 816.638,A 0.000,B 0.000,C 90.000,E1 114.771} C_DIS
LIN {X -0.015,Y -368.925,Z 816.624,A 0.000,B 0.000,C 90.000,E1 112.386} C_DIS
LIN {X -0.156,Y -383.331,Z 816.611,A 0.000,B 0.000,C 90.000,E1 110.066} C_DIS
LIN {X -0.057,Y -399.179,Z 816.599,A 0.000,B 0.000,C 90.000,E1 107.764} C_DIS
LIN {X -0.078,Y -416.582,Z 816.586,A 0.000,B 0.000,C 90.000,E1 105.536} C_DIS
LIN {X 0.006,Y -435.646,Z 816.574,A 0.000,B 0.000,C 90.000,E1 103.355} C_DIS
LIN {X 0.178,Y -455.754,Z 816.563,A 0.000,B 0.000,C 90.000,E1 101.299} C_DIS
LIN {X -0.051,Y -468.460,Z 816.556,A 0.000,B 0.000,C 90.000,E1 100.141} C_DIS
LIN {X -0.096,Y -470.376,Z 816.555,A 0.000,B 0.000,C 90.000,E1 99.905} C_DIS
LIN {X -0.140,Y -471.832,Z 816.554,A 0.000,B 0.000,C 90.000,E1 99.670} C_DIS
LIN {X -0.042,Y -473.819,Z 816.551,A 0.000,B 0.000,C 90.000,E1 99.151} C_DIS
LIN {X 0.141,Y -474.682,Z 816.548,A 0.000,B 0.000,C 90.000,E1 98.624} C_DIS
LIN {X -0.206,Y -474.568,Z 816.545,A 0.000,B 0.000,C 90.000,E1 98.163} C_DIS
LIN {X -0.077,Y -473.466,Z 816.542,A 0.000,B 0.000,C 90.000,E1 97.644} C_DIS
LIN {X -0.216,Y -472.495,Z 816.541,A 0.000,B 0.000,C 90.000,E1 97.409} C_DIS
LIN {X 0.052,Y -471.185,Z 816.540,A 0.000,B 0.000,C 90.000,E1 97.125} C_DIS
LIN {X 0.207,Y -453.535,Z 816.524,A 0.000,B 0.000,C 90.000,E1 94.302} C_DIS
LIN {X -0.098,Y -442.961,Z 816.514,A 0.000,B 0.000,C 90.000,E1 92.522} C_DIS
LIN {X 0.084,Y -433.743,Z 816.505,A 0.000,B 0.000,C 90.000,E1 90.917} C_DIS
LIN {X 0.092,Y -424.156,Z 816.496,A 0.000,B 0.000,C 90.000,E1 89.312} C_DIS
LIN {X -0.056,Y -414.441,Z 816.487,A 0.000,B 0.000,C 90.000,E1 87.707} C_DIS
LIN {X 0.035,Y -404.567,Z 816.478,A 0.000,B 0.000,C 90.000,E1 86.045} C_DIS
LIN {X 0.088,Y -391.391,Z 816.466,A 0.000,B 0.000,C 90.000,E1 83.799} C_DIS
LIN {X -0.097,Y -376.881,Z 816.451,A 0.000,B 0.000,C 90.000,E1 81.254} C_DIS
LIN {X 0.193,Y -362.921,Z 816.437,A 0.000,B 0.000,C 90.000,E1 78.578} C_DIS
LIN {X -0.050,Y -351.092,Z 816.423,A 0.000,B 0.000,C 90.000,E1 76.228} C_DIS
LIN {X -0.062,Y -339.299,Z 816.410,A 0.000,B 0.000,C 90.000,E1 73.795} C_DIS
LIN {X 0.145,Y -327.710,Z 816.396,A 0.000,B 0.000,C 90.000,E1 71.275} C_DIS
LIN {X -0.099,Y -315.017,Z 816.380,A 0.000,B 0.000,C 90.000,E1 68.465} C_DIS
LIN {X -0.143,Y -301.496,Z 816.362,A 0.000,B 0.000,C 90.000,E1 65.229} C_DIS
LIN {X 0.062,Y -291.393,Z 816.347,A 0.000,B 0.000,C 90.000,E1 62.538} C_DIS
LIN {X -0.111,Y -281.617,Z 816.333,A 0.000,B 0.000,C 90.000,E1 59.871} C_DIS
LIN {X -0.013,Y -271.137,Z 816.315,A 0.000,B 0.000,C 90.000,E1 56.755} C_DIS
LIN {X 0.177,Y -262.311,Z 816.300,A 0.000,B 0.000,C 90.000,E1 53.909} C_DIS
LIN {X -0.024,Y -255.794,Z 816.288,A 0.000,B 0.000,C 90.000,E1 51.823} C_DIS
LIN {X -0.153,Y -245.266,Z 816.268,A 0.000,B 0.000,C 90.000,E1 48.243} C_DIS
LIN {X 0.029,Y -235.491,Z 816.247,A 0.000,B 0.000,C 90.000,E1 44.514} C_DIS
LIN {X 0.019,Y -228.278,Z 816.231,A 0.000,B 0.000,C 90.000,E1 41.515} C_DIS
LIN {X 0.040,Y -221.288,Z 816.214,A 0.000,B 0.000,C 90.000,E1 38.463} C_DIS
LIN {X -0.033,Y -214.572,Z 816.197,A 0.000,B 0.000,C 90.000,E1 35.391} C_DIS
LIN {X -0.047,Y -208.256,Z 816.179,A 0.000,B 0.000,C 90.000,E1 32.260} C_DIS
LIN {X -0.024,Y -202.600,Z 816.161,A 0.000,B 0.000,C 90.000,E1 29.077} C_DIS
LIN {X 0.022,Y -197.567,Z 816.144,A 0.000,B 0.000,C 90.000,E1 25.848} C_DIS
LIN {X 0.052,Y -192.444,Z 816.121,A 0.000,B 0.000,C 90.000,E1 21.770} C_DIS
LIN {X -0.069,Y -188.410,Z 816.098,A 0.000,B 0.000,C 90.000,E1 17.692} C_DIS
LIN {X -0.043,Y -185.146,Z 816.070,A 0.000,B 0.000,C 90.000,E1 12.703} C_DIS
LIN {X -0.011,Y -183.049,Z 816.029,A 0.000,B 0.000,C 90.000,E1 5.163} C_DIS
LIN {X 0.071,Y -184.678,Z 815.979,A 0.000,B 0.000,C 90.000,E1 356.159} C_DIS
LIN {X -0.076,Y -187.455,Z 815.951,A 0.000,B 0.000,C 90.000,E1 351.197} C_DIS
LIN {X -0.086,Y -191.460,Z 815.923,A 0.000,B 0.000,C 90.000,E1 346.228} C_DIS
LIN {X -0.108,Y -195.825,Z 815.901,A 0.000,B 0.000,C 90.000,E1 342.127} C_DIS
LIN {X 0.003,Y -201.095,Z 815.878,A 0.000,B 0.000,C 90.000,E1 338.028} C_DIS
LIN {X -0.045,Y -207.220,Z 815.856,A 0.000,B 0.000,C 90.000,E1 334.024} C_DIS
LIN {X -0.031,Y -212.800,Z 815.838,A 0.000,B 0.000,C 90.000,E1 330.845} C_DIS
LIN {X 0.036,Y -220.654,Z 815.816,A 0.000,B 0.000,C 90.000,E1 326.914} C_DIS
LIN {X 0.101,Y -229.300,Z 815.795,A 0.000,B 0.000,C 90.000,E1 323.050} C_DIS
LIN {X 0.024,Y -237.805,Z 815.776,A 0.000,B 0.000,C 90.000,E1 319.666} C_DIS
LIN {X -0.019,Y -247.112,Z 815.757,A 0.000,B 0.000,C 90.000,E1 316.338} C_DIS
LIN {X 0.019,Y -257.316,Z 815.739,A 0.000,B 0.000,C 90.000,E1 313.056} C_DIS
LIN {X 0.009,Y -268.171,Z 815.721,A 0.000,B 0.000,C 90.000,E1 309.850} C_DIS
LIN {X 0.011,Y -279.872,Z 815.704,A 0.000,B 0.000,C 90.000,E1 306.710} C_DIS
LIN {X 0.065,Y -294.322,Z 815.685,A 0.000,B 0.000,C 90.000,E1 303.293} C_DIS
LIN {X -0.052,Y -310.498,Z 815.667,A 0.000,B 0.000,C 90.000,E1 300.001} C_DIS
LIN {X 0.075,Y -326.799,Z 815.651,A 0.000,B 0.000,C 90.000,E1 297.078} C_DIS
LIN {X 0.092,Y -344.519,Z 815.635,A 0.000,B 0.000,C 90.000,E1 294.259} C_DIS
LIN {X -0.112,Y -357.353,Z 815.625,A 0.000,B 0.000,C 90.000,E1 292.461} C_DIS
LIN {X 0.050,Y -375.931,Z 815.612,A 0.000,B 0.000,C 90.000,E1 290.066} C_DIS
LIN {X 0.029,Y -393.530,Z 815.600,A 0.000,B 0.000,C 90.000,E1 288.055} C_DIS
LIN {X -0.028,Y -411.291,Z 815.590,A 0.000,B 0.000,C 90.000,E1 286.134} C_DIS
LIN {X 0.034,Y -423.800,Z 815.582,A 0.000,B 0.000,C 90.000,E1 284.773} C_DIS
LIN {X 0.131,Y -436.131,Z 815.575,A 0.000,B 0.000,C 90.000,E1 283.411} C_DIS
LIN {X 0.086,Y -445.693,Z 815.569,A 0.000,B 0.000,C 90.000,E1 282.355} C_DIS
LIN {X 0.152,Y -454.660,Z 815.563,A 0.000,B 0.000,C 90.000,E1 281.299} C_DIS
LIN {X -0.043,Y -461.005,Z 815.559,A 0.000,B 0.000,C 90.000,E1 280.546} C_DIS
LIN {X 0.121,Y -468.794,Z 815.553,A 0.000,B 0.000,C 90.000,E1 279.500} C_DIS
LIN {X 0.060,Y -474.177,Z 815.549,A 0.000,B 0.000,C 90.000,E1 278.746} C_DIS
LIN {X 0.040,Y -478.953,Z 815.544,A 0.000,B 0.000,C 90.000,E1 277.992} C_DIS
LIN {X 0.063,Y -483.102,Z 815.540,A 0.000,B 0.000,C 90.000,E1 277.239} C_DIS
LIN {X -0.244,Y -485.530,Z 815.537,A 0.000,B 0.000,C 90.000,E1 276.777} C_DIS
LIN {X -0.174,Y -488.553,Z 815.533,A 0.000,B 0.000,C 90.000,E1 276.024} C_DIS
LIN {X -0.020,Y -490.150,Z 815.531,A 0.000,B 0.000,C 90.000,E1 275.511} C_DIS
LIN {X 0.196,Y -491.313,Z 815.528,A 0.000,B 0.000,C 90.000,E1 274.992} C_DIS
LIN {X -0.071,Y -492.133,Z 815.525,A 0.000,B 0.000,C 90.000,E1 274.531} C_DIS
LIN {X 0.157,Y -492.606,Z 815.522,A 0.000,B 0.000,C 90.000,E1 274.012} C_DIS
LIN {X -0.136,Y -492.611,Z 815.520,A 0.000,B 0.000,C 90.000,E1 273.555} C_DIS
LIN {X 0.096,Y -492.299,Z 815.517,A 0.000,B 0.000,C 90.000,E1 273.037} C_DIS
LIN {X -0.190,Y -491.540,Z 815.514,A 0.000,B 0.000,C 90.000,E1 272.579} C_DIS
LIN {X 0.017,Y -490.445,Z 815.511,A 0.000,B 0.000,C 90.000,E1 272.064} C_DIS
LIN {X 0.235,Y -488.903,Z 815.509,A 0.000,B 0.000,C 90.000,E1 271.547} C_DIS
LIN {X -0.058,Y -486.901,Z 815.506,A 0.000,B 0.000,C 90.000,E1 271.088} C_DIS
LIN {X 0.128,Y -484.385,Z 815.503,A 0.000,B 0.000,C 90.000,E1 270.573} C_DIS
LIN {X -0.185,Y -481.207,Z 815.500,A 0.000,B 0.000,C 90.000,E1 270.115} C_DIS
LIN {X -0.032,Y -477.382,Z 815.498,A 0.000,B 0.000,C 90.000,E1 269.599} C_DIS
LIN {X -0.204,Y -475.179,Z 815.496,A 0.000,B 0.000,C 90.000,E1 269.370} C_DIS
LIN {X -0.046,Y -470.008,Z 815.494,A 0.000,B 0.000,C 90.000,E1 268.854} C_DIS
LIN {X -0.092,Y -464.108,Z 815.491,A 0.000,B 0.000,C 90.000,E1 268.396} C_DIS
LIN {X -0.088,Y -457.617,Z 815.489,A 0.000,B 0.000,C 90.000,E1 267.993} C_DIS
LIN {X 0.005,Y -450.511,Z 815.487,A 0.000,B 0.000,C 90.000,E1 267.650} C_DIS
LIN {X 0.203,Y -442.848,Z 815.485,A 0.000,B 0.000,C 90.000,E1 267.364} C_DIS
LIN {X 0.002,Y -435.022,Z 815.484,A 0.000,B 0.000,C 90.000,E1 267.192} C_DIS
LIN {X -0.108,Y -426.990,Z 815.484,A 0.000,B 0.000,C 90.000,E1 267.078} C_DIS
LIN {X -0.094,Y -418.728,Z 815.483,A 0.000,B 0.000,C 90.000,E1 267.020} C_DIS
LIN {X -0.070,Y -180.991,Z 815.483,A 0.000,B 0.000,C 90.000,E1 267.020} C_DIS
LIN {X 0.043,Y -180.854,Z 815.472,A 0.000,B 0.000,C 90.000,E1 264.951} C_DIS
LIN {X -0.082,Y -178.965,Z 815.444,A 0.000,B 0.000,C 90.000,E1 259.926} C_DIS
LIN {X -0.072,Y -177.915,Z 815.435,A 0.000,B 0.000,C 90.000,E1 258.229} C_DIS
LIN {X -0.056,Y -175.550,Z 815.411,A 0.000,B 0.000,C 90.000,E1 253.976} C_DIS
LIN {X -0.049,Y -172.282,Z 815.387,A 0.000,B 0.000,C 90.000,E1 249.699} C_DIS
LIN {X -0.009,Y -171.761,Z 815.382,A 0.000,B 0.000,C 90.000,E1 248.827} C_DIS
LIN {X 0.008,Y -167.361,Z 815.354,A 0.000,B 0.000,C 90.000,E1 243.640} C_DIS
LIN {X 0.090,Y -166.749,Z 815.349,A 0.000,B 0.000,C 90.000,E1 242.743} C_DIS
LIN {X 0.002,Y -162.729,Z 815.324,A 0.000,B 0.000,C 90.000,E1 238.408} C_DIS
LIN {X 0.063,Y -161.420,Z 815.315,A 0.000,B 0.000,C 90.000,E1 236.628} C_DIS
LIN {X 0.104,Y -157.413,Z 815.290,A 0.000,B 0.000,C 90.000,E1 232.190} C_DIS
LIN {X 0.036,Y -155.414,Z 815.275,A 0.000,B 0.000,C 90.000,E1 229.542} C_DIS
LIN {X -0.033,Y -151.742,Z 815.250,A 0.000,B 0.000,C 90.000,E1 225.081} C_DIS
LIN {X -0.020,Y -149.939,Z 815.235,A 0.000,B 0.000,C 90.000,E1 222.366} C_DIS
LIN {X 0.007,Y -146.787,Z 815.210,A 0.000,B 0.000,C 90.000,E1 217.810} C_DIS
LIN {X -0.092,Y -145.360,Z 815.195,A 0.000,B 0.000,C 90.000,E1 215.105} C_DIS
LIN {X 0.025,Y -142.429,Z 815.164,A 0.000,B 0.000,C 90.000,E1 209.539} C_DIS
LIN {X 0.075,Y -141.417,Z 815.149,A 0.000,B 0.000,C 90.000,E1 206.744} C_DIS
LIN {X 0.061,Y -139.361,Z 815.113,A 0.000,B 0.000,C 90.000,E1 200.248} C_DIS
LIN {X 0.048,Y -138.804,Z 815.097,A 0.000,B 0.000,C 90.000,E1 197.457} C_DIS
LIN {X -0.032,Y -138.350,Z 815.056,A 0.000,B 0.000,C 90.000,E1 190.018} C_DIS
LIN {X -0.057,Y -139.545,Z 815.004,A 0.000,B 0.000,C 90.000,E1 180.688} C_DIS
LIN {X 0.035,Y -141.249,Z 814.973,A 0.000,B 0.000,C 90.000,E1 175.065} C_DIS
LIN {X -0.006,Y -142.618,Z 814.957,A 0.000,B 0.000,C 90.000,E1 172.299} C_DIS
LIN {X -0.053,Y -144.936,Z 814.932,A 0.000,B 0.000,C 90.000,E1 167.701} C_DIS
LIN {X 0.080,Y -147.564,Z 814.911,A 0.000,B 0.000,C 90.000,E1 163.976} C_DIS
LIN {X -0.031,Y -150.172,Z 814.891,A 0.000,B 0.000,C 90.000,E1 160.369} C_DIS
LIN {X -0.022,Y -153.546,Z 814.871,A 0.000,B 0.000,C 90.000,E1 156.741} C_DIS
LIN {X 0.030,Y -156.964,Z 814.851,A 0.000,B 0.000,C 90.000,E1 153.127} C_DIS
LIN {X -0.035,Y -161.073,Z 814.831,A 0.000,B 0.000,C 90.000,E1 149.587} C_DIS
LIN {X 0.050,Y -163.180,Z 814.821,A 0.000,B 0.000,C 90.000,E1 147.788} C_DIS
LIN {X 0.056,Y -167.601,Z 814.802,A 0.000,B 0.000,C 90.000,E1 144.276} C_DIS
LIN {X -0.035,Y -171.429,Z 814.787,A 0.000,B 0.000,C 90.000,E1 141.698} C_DIS
LIN {X 0.004,Y -176.349,Z 814.768,A 0.000,B 0.000,C 90.000,E1 138.243} C_DIS
LIN {X 0.001,Y -180.639,Z 814.754,A 0.000,B 0.000,C 90.000,E1 135.688} C_DIS
LIN {X -0.015,Y -186.041,Z 814.735,A 0.000,B 0.000,C 90.000,E1 132.324} C_DIS
LIN {X 0.048,Y -190.676,Z 814.721,A 0.000,B 0.000,C 90.000,E1 129.806} C_DIS
LIN {X -0.011,Y -192.733,Z 814.714,A 0.000,B 0.000,C 90.000,E1 128.588} C_DIS
LIN {X -0.050,Y -293.281,Z 814.714,A 0.000,B 0.000,C 90.000,E1 128.588} C_DIS
LIN {X -0.027,Y -295.266,Z 814.714,A 0.000,B 0.000,C 90.000,E1 128.543} C_DIS
LIN {X -0.152,Y -299.051,Z 814.713,A 0.000,B 0.000,C 90.000,E1 128.382} C_DIS
LIN {X -0.044,Y -301.309,Z 814.712,A 0.000,B 0.000,C 90.000,E1 128.177} C_DIS
LIN {X 0.012,Y -305.172,Z 814.709,A 0.000,B 0.000,C 90.000,E1 127.684} C_DIS
LIN {X -0.035,Y -307.000,Z 814.708,A 0.000,B 0.000,C 90.000,E1 127.363} C_DIS
LIN {X -0.024,Y -308.426,Z 814.706,A 0.000,B 0.000,C 90.000,E1 127.030} C_DIS
LIN {X -0.025,Y -310.472,Z 814.702,A 0.000,B 0.000,C 90.000,E1 126.377} C_DIS
LIN {X -0.144,Y -320.596,Z 814.684,A 0.000,B 0.000,C 90.000,E1 123.166} C_DIS
LIN {X 0.154,Y -331.029,Z 814.668,A 0.000,B 0.000,C 90.000,E1 120.256} C_DIS
LIN {X 0.095,Y -342.818,Z 814.653,A 0.000,B 0.000,C 90.000,E1 117.462} C_DIS
LIN {X 0.073,Y -356.063,Z 814.637,A 0.000,B 0.000,C 90.000,E1 114.719} C_DIS
LIN {X 0.040,Y -369.157,Z 814.624,A 0.000,B 0.000,C 90.000,E1 112.333} C_DIS
LIN {X 0.046,Y -383.590,Z 814.611,A 0.000,B 0.000,C 90.000,E1 109.993} C_DIS
LIN {X 0.150,Y -399.465,Z 814.598,A 0.000,B 0.000,C 90.000,E1 107.692} C_DIS
LIN {X 0.022,Y -416.898,Z 814.586,A 0.000,B 0.000,C 90.000,E1 105.481} C_DIS
LIN {X 0.125,Y -435.992,Z 814.574,A 0.000,B 0.000,C 90.000,E1 103.300} C_DIS
LIN {X -0.115,Y -456.111,Z 814.563,A 0.000,B 0.000,C 90.000,E1 101.299} C_DIS
LIN {X 0.183,Y -466.379,Z 814.557,A 0.000,B 0.000,C 90.000,E1 100.310} C_DIS
LIN {X 0.206,Y -468.750,Z 814.556,A 0.000,B 0.000,C 90.000,E1 100.074} C_DIS
LIN {X 0.047,Y -470.623,Z 814.555,A 0.000,B 0.000,C 90.000,E1 99.849} C_DIS
LIN {X -0.032,Y -472.041,Z 814.553,A 0.000,B 0.000,C 90.000,E1 99.613} C_DIS
LIN {X 0.070,Y -473.928,Z 814.551,A 0.000,B 0.000,C 90.000,E1 99.095} C_DIS
LIN {X -0.215,Y -474.709,Z 814.548,A 0.000,B 0.000,C 90.000,E1 98.624} C_DIS
LIN {X -0.092,Y -474.519,Z 814.545,A 0.000,B 0.000,C 90.000,E1 98.106} C_DIS
LIN {X 0.038,Y -473.333,Z 814.542,A 0.000,B 0.000,C 90.000,E1 97.587} C_DIS
LIN {X -0.102,Y -472.312,Z 814.541,A 0.000,B 0.000,C 90.000,E1 97.352} C_DIS
LIN {X 0.166,Y -470.940,Z 814.539,A 0.000,B 0.000,C 90.000,E1 97.068} C_DIS
LIN {X -0.140,Y -453.301,Z 814.524,A 0.000,B 0.000,C 90.000,E1 94.302} C_DIS
LIN {X 0.001,Y -442.720,Z 814.514,A 0.000,B 0.000,C 90.000,E1 92.465} C_DIS
LIN {X 0.176,Y -433.515,Z 814.505,A 0.000,B 0.000,C 90.000,E1 90.859} C_DIS
LIN {X 0.179,Y -423.928,Z 814.496,A 0.000,B 0.000,C 90.000,E1 89.255} C_DIS
LIN {X 0.114,Y -412.574,Z 814.485,A 0.000,B 0.000,C 90.000,E1 87.364} C_DIS
LIN {X 0.194,Y -402.675,Z 814.476,A 0.000,B 0.000,C 90.000,E1 85.698} C_DIS
LIN {X 0.161,Y -389.534,Z 814.464,A 0.000,B 0.000,C 90.000,E1 83.457} C_DIS
LIN {X -0.023,Y -375.126,Z 814.449,A 0.000,B 0.000,C 90.000,E1 80.905} C_DIS
LIN {X -0.170,Y -359.715,Z 814.433,A 0.000,B 0.000,C 90.000,E1 77.993} C_DIS
LIN {X -0.055,Y -347.965,Z 814.420,A 0.000,B 0.000,C 90.000,E1 75.574} C_DIS
LIN {X -0.143,Y -336.242,Z 814.406,A 0.000,B 0.000,C 90.000,E1 73.142} C_DIS
LIN {X 0.092,Y -324.723,Z 814.392,A 0.000,B 0.000,C 90.000,E1 70.604} C_DIS
LIN {X 0.059,Y -312.168,Z 814.376,A 0.000,B 0.000,C 90.000,E1 67.741} C_DIS
LIN {X 0.046,Y -297.624,Z 814.356,A 0.000,B 0.000,C 90.000,E1 64.152} C_DIS
LIN {X -0.130,Y -286.483,Z 814.340,A 0.000,B 0.000,C 90.000,E1 61.179} C_DIS
LIN {X -0.003,Y -274.695,Z 814.321,A 0.000,B 0.000,C 90.000,E1 57.740} C_DIS
LIN {X -0.031,Y -264.637,Z 814.303,A 0.000,B 0.000,C 90.000,E1 54.609} C_DIS
LIN {X 0.015,Y -258.150,Z 814.292,A 0.000,B 0.000,C 90.000,E1 52.477} C_DIS
LIN {X -0.050,Y -249.578,Z 814.276,A 0.000,B 0.000,C 90.000,E1 49.622} C_DIS
LIN {X -0.070,Y -239.489,Z 814.255,A 0.000,B 0.000,C 90.000,E1 45.972} C_DIS
LIN {X -0.064,Y -230.275,Z 814.235,A 0.000,B 0.000,C 90.000,E1 42.243} C_DIS
LIN {X -0.013,Y -223.265,Z 814.218,A 0.000,B 0.000,C 90.000,E1 39.197} C_DIS
LIN {X 0.103,Y -214.794,Z 814.196,A 0.000,B 0.000,C 90.000,E1 35.311} C_DIS
LIN {X -0.025,Y -208.488,Z 814.179,A 0.000,B 0.000,C 90.000,E1 32.212} C_DIS
LIN {X 0.010,Y -202.847,Z 814.161,A 0.000,B 0.000,C 90.000,E1 29.027} C_DIS
LIN {X 0.066,Y -197.826,Z 814.143,A 0.000,B 0.000,C 90.000,E1 25.796} C_DIS
LIN {X -0.071,Y -192.695,Z 814.121,A 0.000,B 0.000,C 90.000,E1 21.770} C_DIS
LIN {X -0.002,Y -188.664,Z 814.098,A 0.000,B 0.000,C 90.000,E1 17.638} C_DIS
LIN {X 0.036,Y -185.425,Z 814.070,A 0.000,B 0.000,C 90.000,E1 12.647} C_DIS
LIN {X 0.086,Y -183.307,Z 814.029,A 0.000,B 0.000,C 90.000,E1 5.106} C_DIS
LIN {X 0.078,Y -184.936,Z 813.979,A 0.000,B 0.000,C 90.000,E1 356.159} C_DIS
LIN {X -0.060,Y -187.690,Z 813.951,A 0.000,B 0.000,C 90.000,E1 351.197} C_DIS
LIN {X -0.062,Y -191.664,Z 813.923,A 0.000,B 0.000,C 90.000,E1 346.228} C_DIS
LIN {X -0.077,Y -196.011,Z 813.901,A 0.000,B 0.000,C 90.000,E1 342.127} C_DIS
LIN {X 0.041,Y -201.245,Z 813.878,A 0.000,B 0.000,C 90.000,E1 338.028} C_DIS
LIN {X -0.001,Y -207.371,Z 813.856,A 0.000,B 0.000,C 90.000,E1 334.024} C_DIS
